LIN {X 0,Y 175.401,Z 600.795,A -85,B 0,C 180,E1 -24078.805,E2 -24078.805} C_VEL
LIN {X 0,Y 170.127,Z 592.607,A -85,B 0,C 180,E1 -24081.433,E2 -24081.433} C_VEL
LIN {X 0,Y 165.142,Z 585.432,A -85,B 0,C 180,E1 -24084.194,E2 -24084.194} C_VEL
LIN {X 0,Y 162.074,Z 581.252,A -85,B 0,C 180,E1 -24086.061,E2 -24086.061} C_VEL
LIN {X 0,Y 159.438,Z 578,A -85,B 0,C 180,E1 -24087.775,E2 -24087.775} C_VEL
LIN {X 0,Y 158.547,Z 576.618,A -85,B 0,C 180,E1 -24088.411,E2 -24088.411} C_VEL
LIN {X 0,Y 155.998,Z 573.951,A -85,B 0,C 180,E1 -24090.222,E2 -24090.222} C_VEL
LIN {X 0,Y 154.688,Z 571.494,A -85,B 0,C 180,E1 -24091.321,E2 -24091.321} C_VEL
LIN {X 0,Y 152.117,Z 569.719,A -85,B 0,C 180,E1 -24093.343,E2 -24093.343} C_VEL
LIN {X 0,Y 150.618,Z 567.322,A -85,B 0,C 180,E1 -24094.775,E2 -24094.775} C_VEL
LIN {X 0,Y 150.248,Z 565.769,A -85,B 0,C 180,E1 -24095.287,E2 -24095.287} C_VEL
LIN {X 0,Y 150.36,Z 565.755,A -85,B 0,C 180,E1 -24100.902,E2 -24100.902} C_VEL
LIN {X 0,Y 150.448,Z 565.742,A -85,B 0,C 180,E1 -24106.493,E2 -24106.493} C_VEL
LIN {X 0,Y 150.645,Z 565.698,A -85,B 0,C 180,E1 -24109.245,E2 -24109.245} C_VEL
LIN {X 0,Y 150.739,Z 565.693,A -85,B 0,C 180,E1 -24111.959,E2 -24111.959} C_VEL
LIN {X 0,Y 151.214,Z 565.649,A -85,B 0,C 180,E1 -24120,E2 -24120} C_VEL
LIN {X 0,Y 150.757,Z 565.696,A -85,B 0,C 180,E1 -24128.039,E2 -24128.039} C_VEL
LIN {X 0,Y 150.628,Z 565.705,A -85,B 0,C 180,E1 -24131.545,E2 -24131.545} C_VEL
LIN {X 0,Y 150.369,Z 565.735,A -85,B 0,C 180,E1 -24136.286,E2 -24136.286} C_VEL
LIN {X 0,Y 150.346,Z 565.743,A -85,B 0,C 180,E1 -24140.794,E2 -24140.794} C_VEL
LIN {X 0,Y 150.251,Z 565.771,A -85,B 0,C 180,E1 -24144.343,E2 -24144.343} C_VEL
LIN {X 0,Y 150.963,Z 568.144,A -85,B 0,C 180,E1 -24145.232,E2 -24145.232} C_VEL
LIN {X 0,Y 152.896,Z 570.41,A -85,B 0,C 180,E1 -24146.946,E2 -24146.946} C_VEL
LIN {X 0,Y 154.763,Z 571.667,A -85,B 0,C 180,E1 -24148.385,E2 -24148.385} C_VEL
LIN {X 0,Y 156.509,Z 574.692,A -85,B 0,C 180,E1 -24149.812,E2 -24149.812} C_VEL
LIN {X 0,Y 158.954,Z 577.113,A -85,B 0,C 180,E1 -24151.509,E2 -24151.509} C_VEL
LIN {X 0,Y 161.394,Z 580.608,A -85,B 0,C 180,E1 -24153.164,E2 -24153.164} C_VEL
LIN {X 0,Y 162.927,Z 582.356,A -85,B 0,C 180,E1 -24154.109,E2 -24154.109} C_VEL
LIN {X 0,Y 166.851,Z 588.676,A -85,B 0,C 180,E1 -24156.487,E2 -24156.487} C_VEL
LIN {X 0,Y 171.487,Z 596.616,A -85,B 0,C 180,E1 -24159.037,E2 -24159.037} C_VEL
LIN {X 0,Y 177.334,Z 608.087,A -85,B 0,C 180,E1 -24161.98,E2 -24161.98} C_VEL
LIN {X 0,Y 182.328,Z 619.835,A -85,B 0,C 180,E1 -24164.336,E2 -24164.336} C_VEL
LIN {X 0,Y 185.647,Z 628.738,A -85,B 0,C 180,E1 -24165.839,E2 -24165.839} C_VEL
LIN {X 0,Y 185.583,Z 633.595,A -85,B 0,C 180,E1 -24166.075,E2 -24166.075} C_VEL
LIN {X 0,Y 182.946,Z 673.813,A -85,B 0,C 180,E1 -24167.507,E2 -24167.507} C_VEL
LIN {X 0,Y 181.015,Z 687.597,A -85,B 0,C 180,E1 -24168.363,E2 -24168.363} C_VEL
LIN {X 0,Y 178.414,Z 699.716,A -85,B 0,C 180,E1 -24169.464,E2 -24169.464} C_VEL
LIN {X 0,Y 174.982,Z 712.384,A -85,B 0,C 180,E1 -24171.132,E2 -24171.132} C_VEL
LIN {X 0,Y 171.291,Z 723.647,A -85,B 0,C 180,E1 -24173.129,E2 -24173.129} C_VEL
LIN {X 0,Y 167.361,Z 733.791,A -85,B 0,C 180,E1 -24175.468,E2 -24175.468} C_VEL
LIN {X 0,Y 163.41,Z 742.938,A -85,B 0,C 180,E1 -24178.21,E2 -24178.21} C_VEL
LIN {X 0,Y 161.853,Z 746.354,A -85,B 0,C 180,E1 -24179.425,E2 -24179.425} C_VEL
LIN {X 0,Y 159.445,Z 750.159,A -85,B 0,C 180,E1 -24180.827,E2 -24180.827} C_VEL
LIN {X 0,Y 154.006,Z 755.881,A -85,B 0,C 180,E1 -24183.055,E2 -24183.055} C_VEL
LIN {X 0,Y 148.739,Z 760.905,A -85,B 0,C 180,E1 -24185.589,E2 -24185.589} C_VEL
LIN {X 0,Y 146.663,Z 763.652,A -85,B 0,C 180,E1 -24187.435,E2 -24187.435} C_VEL
LIN {X 0,Y 144.028,Z 768.399,A -85,B 0,C 180,E1 -24191.511,E2 -24191.511} C_VEL
LIN {X 0,Y 142.223,Z 772.01,A -85,B 0,C 180,E1 -24195.698,E2 -24195.698} C_VEL
LIN {X 0,Y 141.401,Z 773.873,A -85,B 0,C 180,E1 -24198.535,E2 -24198.535} C_VEL
LIN {X 0,Y 140.849,Z 775.27,A -85,B 0,C 180,E1 -24201.393,E2 -24201.393} C_VEL
LIN {X 0,Y 140.554,Z 776.27,A -85,B 0,C 180,E1 -24204.263,E2 -24204.263} C_VEL
LIN {X 0,Y 140.562,Z 777.087,A -85,B 0,C 180,E1 -24209.713,E2 -24209.713} C_VEL
LIN {X 0,Y 140.736,Z 776.871,A -85,B 0,C 180,E1 -24212.865,E2 -24212.865} C_VEL
LIN {X 0,Y 141.065,Z 776.256,A -85,B 0,C 180,E1 -24215.721,E2 -24215.721} C_VEL
LIN {X 0,Y 141.616,Z 775.252,A -85,B 0,C 180,E1 -24218.565,E2 -24218.565} C_VEL
LIN {X 0,Y 144.026,Z 772.019,A -85,B 0,C 180,E1 -24224.395,E2 -24224.395} C_VEL
LIN {X 0,Y 146.516,Z 776.665,A -85,B 0,C 180,E1 -24229.622,E2 -24229.622} C_VEL
LIN {X 0,Y 148.4,Z 778.596,A -85,B 0,C 180,E1 -24232.266,E2 -24232.266} C_VEL
LIN {X 0,Y 153.432,Z 781.157,A -85,B 0,C 180,E1 -24237.264,E2 -24237.264} C_VEL
LIN {X 0,Y 156.692,Z 781.963,A -85,B 0,C 180,E1 -24239.565,E2 -24239.565} C_VEL
LIN {X 0,Y 164.15,Z 782.273,A -85,B 0,C 180,E1 -24243.822,E2 -24243.822} C_VEL
LIN {X 0,Y 168.36,Z 781.919,A -85,B 0,C 180,E1 -24245.764,E2 -24245.764} C_VEL
LIN {X 0,Y 177.623,Z 779.864,A -85,B 0,C 180,E1 -24249.279,E2 -24249.279} C_VEL
LIN {X 0,Y 185.169,Z 777.289,A -85,B 0,C 180,E1 -24251.623,E2 -24251.623} C_VEL
LIN {X 0,Y 193.201,Z 773.68,A -85,B 0,C 180,E1 -24253.724,E2 -24253.724} C_VEL
LIN {X 0,Y 198.847,Z 770.696,A -85,B 0,C 180,E1 -24254.983,E2 -24254.983} C_VEL
LIN {X 0,Y 201.924,Z 768.865,A -85,B 0,C 180,E1 -24255.885,E2 -24255.885} C_VEL
LIN {X 0,Y 193.405,Z 773.579,A -85,B 0,C 180,E1 -24257.758,E2 -24257.758} C_VEL
LIN {X 0,Y 185.332,Z 777.13,A -85,B 0,C 180,E1 -24259.86,E2 -24259.86} C_VEL
LIN {X 0,Y 175.364,Z 780.219,A -85,B 0,C 180,E1 -24263.048,E2 -24263.048} C_VEL
LIN {X 0,Y 170.717,Z 781.07,A -85,B 0,C 180,E1 -24264.806,E2 -24264.806} C_VEL
LIN {X 0,Y 162.284,Z 781.531,A -85,B 0,C 180,E1 -24268.689,E2 -24268.689} C_VEL
LIN {X 0,Y 158.606,Z 781.187,A -85,B 0,C 180,E1 -24270.829,E2 -24270.829} C_VEL
LIN {X 0,Y 152.19,Z 779.18,A -85,B 0,C 180,E1 -24275.442,E2 -24275.442} C_VEL
LIN {X 0,Y 148.495,Z 776.67,A -85,B 0,C 180,E1 -24279.209,E2 -24279.209} C_VEL
LIN {X 0,Y 145.778,Z 773.203,A -85,B 0,C 180,E1 -24283.186,E2 -24283.186} C_VEL
LIN {X 0,Y 144.118,Z 768.862,A -85,B 0,C 180,E1 -24287.25,E2 -24287.25} C_VEL
LIN {X 0,Y 143.374,Z 764.179,A -85,B 0,C 180,E1 -24290.833,E2 -24290.833} C_VEL
LIN {X 0,Y 143.375,Z 757.493,A -85,B 0,C 180,E1 -24295.079,E2 -24295.079} C_VEL
LIN {X 0,Y 143.685,Z 750.494,A -85,B 0,C 180,E1 -24298.599,E2 -24298.599} C_VEL
LIN {X 0,Y 144.031,Z 742.449,A -85,B 0,C 180,E1 -24301.748,E2 -24301.748} C_VEL
LIN {X 0,Y 144.283,Z 733.555,A -85,B 0,C 180,E1 -24304.54,E2 -24304.54} C_VEL
LIN {X 0,Y 144.601,Z 723.972,A -85,B 0,C 180,E1 -24306.979,E2 -24306.979} C_VEL
LIN {X 0,Y 145.094,Z 712.443,A -85,B 0,C 180,E1 -24309.233,E2 -24309.233} C_VEL
LIN {X 0,Y 145.364,Z 701.518,A -85,B 0,C 180,E1 -24310.798,E2 -24310.798} C_VEL
LIN {X 0,Y 145.916,Z 666.157,A -85,B 0,C 180,E1 -24314.417,E2 -24314.417} C_VEL
LIN {X 0,Y 146.086,Z 645.484,A -85,B 0,C 180,E1 -24316.421,E2 -24316.421} C_VEL
LIN {X 0,Y 144.453,Z 621.674,A -85,B 0,C 180,E1 -24318.574,E2 -24318.574} C_VEL
LIN {X 0,Y 144.39,Z 617.741,A -85,B 0,C 180,E1 -24318.996,E2 -24318.996} C_VEL
LIN {X 0,Y 145.352,Z 604.834,A -85,B 0,C 180,E1 -24323.849,E2 -24323.849} C_VEL
LIN {X 0,Y 145.798,Z 602.705,A -85,B 0,C 180,E1 -24325.137,E2 -24325.137} C_VEL
LIN {X 0,Y 146.091,Z 602.477,A -85,B 0,C 180,E1 -24325.656,E2 -24325.656} C_VEL
LIN {X 0,Y 147.528,Z 602.404,A -85,B 0,C 180,E1 -24326.909,E2 -24326.909} C_VEL
LIN {X 0,Y 150.097,Z 600.201,A -85,B 0,C 180,E1 -24328.582,E2 -24328.582} C_VEL
LIN {X 0,Y 154.19,Z 595.325,A -85,B 0,C 180,E1 -24330.849,E2 -24330.849} C_VEL
LIN {X 0,Y 156.922,Z 595.505,A -85,B 0,C 180,E1 -24332.51,E2 -24332.51} C_VEL
LIN {X 0,Y 158.927,Z 594.524,A -85,B 0,C 180,E1 -24333.557,E2 -24333.557} C_VEL
LIN {X 0,Y 162.927,Z 594.201,A -85,B 0,C 180,E1 -24335.615,E2 -24335.615} C_VEL
LIN {X 0,Y 164.092,Z 594.078,A -85,B 0,C 180,E1 -24336.175,E2 -24336.175} C_VEL
LIN {X 0,Y 168.438,Z 600.642,A -85,B 0,C 180,E1 -24338.61,E2 -24338.61} C_VEL
LIN {X 0,Y 174.079,Z 610.004,A -85,B 0,C 180,E1 -24341.474,E2 -24341.474} C_VEL
LIN {X 0,Y 178.176,Z 617.897,A -85,B 0,C 180,E1 -24343.412,E2 -24343.412} C_VEL
LIN {X 0,Y 180.855,Z 624.585,A -85,B 0,C 180,E1 -24344.681,E2 -24344.681} C_VEL
LIN {X 0,Y 178.238,Z 663.283,A -85,B 0,C 180,E1 -24346.03,E2 -24346.03} C_VEL
LIN {X 0,Y 176.727,Z 676.165,A -85,B 0,C 180,E1 -24346.773,E2 -24346.773} C_VEL
LIN {X 0,Y 174.414,Z 688.968,A -85,B 0,C 180,E1 -24347.938,E2 -24347.938} C_VEL
LIN {X 0,Y 171.475,Z 700.769,A -85,B 0,C 180,E1 -24349.407,E2 -24349.407} C_VEL
LIN {X 0,Y 168.109,Z 711.495,A -85,B 0,C 180,E1 -24351.162,E2 -24351.162} C_VEL
LIN {X 0,Y 164.039,Z 722.429,A -85,B 0,C 180,E1 -24353.524,E2 -24353.524} C_VEL
LIN {X 0,Y 160.287,Z 731.314,A -85,B 0,C 180,E1 -24356.009,E2 -24356.009} C_VEL
LIN {X 0,Y 156.293,Z 739.948,A -85,B 0,C 180,E1 -24359.106,E2 -24359.106} C_VEL
LIN {X 0,Y 152.499,Z 747.445,A -85,B 0,C 180,E1 -24362.555,E2 -24362.555} C_VEL
LIN {X 0,Y 148.926,Z 753.853,A -85,B 0,C 180,E1 -24366.349,E2 -24366.349} C_VEL
LIN {X 0,Y 146.044,Z 758.933,A -85,B 0,C 180,E1 -24370.312,E2 -24370.312} C_VEL
LIN {X 0,Y 143.747,Z 762.872,A -85,B 0,C 180,E1 -24374.399,E2 -24374.399} C_VEL
LIN {X 0,Y 142.139,Z 765.777,A -85,B 0,C 180,E1 -24378.591,E2 -24378.591} C_VEL
LIN {X 0,Y 141.435,Z 767.165,A -85,B 0,C 180,E1 -24381.424,E2 -24381.424} C_VEL
LIN {X 0,Y 141.008,Z 768.151,A -85,B 0,C 180,E1 -24384.277,E2 -24384.277} C_VEL
LIN {X 0,Y 140.737,Z 768.758,A -85,B 0,C 180,E1 -24387.135,E2 -24387.135} C_VEL
LIN {X 0,Y 140.69,Z 768.984,A -85,B 0,C 180,E1 -24389.998,E2 -24389.998} C_VEL
LIN {X 0,Y 140.736,Z 768.789,A -85,B 0,C 180,E1 -24392.86,E2 -24392.86} C_VEL
LIN {X 0,Y 141.007,Z 768.204,A -85,B 0,C 180,E1 -24395.718,E2 -24395.718} C_VEL
LIN {X 0,Y 142.136,Z 765.884,A -85,B 0,C 180,E1 -24401.405,E2 -24401.405} C_VEL
LIN {X 0,Y 143.73,Z 763.013,A -85,B 0,C 180,E1 -24405.598,E2 -24405.598} C_VEL
LIN {X 0,Y 145.977,Z 759.117,A -85,B 0,C 180,E1 -24409.692,E2 -24409.692} C_VEL
LIN {X 0,Y 148.832,Z 754.096,A -85,B 0,C 180,E1 -24413.662,E2 -24413.662} C_VEL
LIN {X 0,Y 152.426,Z 747.763,A -85,B 0,C 180,E1 -24417.454,E2 -24417.454} C_VEL
LIN {X 0,Y 156.142,Z 740.567,A -85,B 0,C 180,E1 -24420.801,E2 -24420.801} C_VEL
LIN {X 0,Y 160.206,Z 731.769,A -85,B 0,C 180,E1 -24424.006,E2 -24424.006} C_VEL
LIN {X 0,Y 164.362,Z 721.91,A -85,B 0,C 180,E1 -24426.769,E2 -24426.769} C_VEL
LIN {X 0,Y 168.516,Z 710.802,A -85,B 0,C 180,E1 -24429.105,E2 -24429.105} C_VEL
LIN {X 0,Y 171.87,Z 699.908,A -85,B 0,C 180,E1 -24430.861,E2 -24430.861} C_VEL
LIN {X 0,Y 174.791,Z 687.856,A -85,B 0,C 180,E1 -24432.334,E2 -24432.334} C_VEL
LIN {X 0,Y 177.054,Z 675.297,A -85,B 0,C 180,E1 -24433.42,E2 -24433.42} C_VEL
LIN {X 0,Y 178.514,Z 662.659,A -85,B 0,C 180,E1 -24434.119,E2 -24434.119} C_VEL
LIN {X 0,Y 181.017,Z 624.787,A -85,B 0,C 180,E1 -24435.451,E2 -24435.451} C_VEL
LIN {X 0,Y 177.262,Z 615.769,A -85,B 0,C 180,E1 -24437.232,E2 -24437.232} C_VEL
LIN {X 0,Y 171.522,Z 605.541,A -85,B 0,C 180,E1 -24440.013,E2 -24440.013} C_VEL
LIN {X 0,Y 166.095,Z 596.948,A -85,B 0,C 180,E1 -24442.917,E2 -24442.917} C_VEL
LIN {X 0,Y 161.753,Z 590.618,A -85,B 0,C 180,E1 -24445.502,E2 -24445.502} C_VEL
LIN {X 0,Y 159.087,Z 586.942,A -85,B 0,C 180,E1 -24447.236,E2 -24447.236} C_VEL
LIN {X 0,Y 156.431,Z 583.249,A -85,B 0,C 180,E1 -24449.115,E2 -24449.115} C_VEL
LIN {X 0,Y 153.386,Z 579.692,A -85,B 0,C 180,E1 -24451.429,E2 -24451.429} C_VEL
LIN {X 0,Y 152.306,Z 577.95,A -85,B 0,C 180,E1 -24452.364,E2 -24452.364} C_VEL
LIN {X 0,Y 149.696,Z 575.629,A -85,B 0,C 180,E1 -24454.609,E2 -24454.609} C_VEL
LIN {X 0,Y 148.169,Z 572.834,A -85,B 0,C 180,E1 -24456.223,E2 -24456.223} C_VEL
LIN {X 0,Y 147.867,Z 572.411,A -85,B 0,C 180,E1 -24456.543,E2 -24456.543} C_VEL
LIN {X 0,Y 145.469,Z 570.902,A -85,B 0,C 180,E1 -24459.052,E2 -24459.052} C_VEL
LIN {X 0,Y 143.833,Z 568.534,A -85,B 0,C 180,E1 -24461.205,E2 -24461.205} C_VEL
LIN {X 0,Y 143.277,Z 566.62,A -85,B 0,C 180,E1 -24462.331,E2 -24462.331} C_VEL
LIN {X 0,Y 143.588,Z 566.58,A -85,B 0,C 180,E1 -24468.709,E2 -24468.709} C_VEL
LIN {X 0,Y 143.659,Z 566.571,A -85,B 0,C 180,E1 -24471.56,E2 -24471.56} C_VEL
LIN {X 0,Y 144.172,Z 566.526,A -85,B 0,C 180,E1 -24480,E2 -24480} C_VEL
LIN {X 0,Y 143.679,Z 566.573,A -85,B 0,C 180,E1 -24488.438,E2 -24488.438} C_VEL
LIN {X 0,Y 143.565,Z 566.586,A -85,B 0,C 180,E1 -24491.758,E2 -24491.758} C_VEL
LIN {X 0,Y 143.287,Z 566.71,A -85,B 0,C 180,E1 -24497.483,E2 -24497.483} C_VEL
LIN {X 0,Y 143.994,Z 568.91,A -85,B 0,C 180,E1 -24498.681,E2 -24498.681} C_VEL
LIN {X 0,Y 145.834,Z 571.244,A -85,B 0,C 180,E1 -24501.008,E2 -24501.008} C_VEL
LIN {X 0,Y 148.092,Z 572.649,A -85,B 0,C 180,E1 -24503.326,E2 -24503.326} C_VEL
LIN {X 0,Y 149.662,Z 575.608,A -85,B 0,C 180,E1 -24505.001,E2 -24505.001} C_VEL
LIN {X 0,Y 152.592,Z 578.316,A -85,B 0,C 180,E1 -24507.517,E2 -24507.517} C_VEL
LIN {X 0,Y 154.86,Z 581.681,A -85,B 0,C 180,E1 -24509.387,E2 -24509.387} C_VEL
LIN {X 0,Y 156.547,Z 583.501,A -85,B 0,C 180,E1 -24510.618,E2 -24510.618} C_VEL
LIN {X 0,Y 159.281,Z 587.171,A -85,B 0,C 180,E1 -24512.531,E2 -24512.531} C_VEL
LIN {X 0,Y 161.27,Z 590.153,A -85,B 0,C 180,E1 -24513.848,E2 -24513.848} C_VEL
LIN {X 0,Y 165.359,Z 596.983,A -85,B 0,C 180,E1 -24516.384,E2 -24516.384} C_VEL
LIN {X 0,Y 170.544,Z 606.852,A -85,B 0,C 180,E1 -24519.316,E2 -24519.316} C_VEL
LIN {X 0,Y 175.099,Z 616.732,A -85,B 0,C 180,E1 -24521.689,E2 -24521.689} C_VEL
LIN {X 0,Y 179.891,Z 629.091,A -85,B 0,C 180,E1 -24524.062,E2 -24524.062} C_VEL
LIN {X 0,Y 180.657,Z 631.538,A -85,B 0,C 180,E1 -24524.447,E2 -24524.447} C_VEL
LIN {X 0,Y 177.817,Z 673.249,A -85,B 0,C 180,E1 -24525.942,E2 -24525.942} C_VEL
LIN {X 0,Y 175.897,Z 686.736,A -85,B 0,C 180,E1 -24526.778,E2 -24526.778} C_VEL
LIN {X 0,Y 173.072,Z 699.517,A -85,B 0,C 180,E1 -24527.934,E2 -24527.934} C_VEL
LIN {X 0,Y 169.524,Z 712.185,A -85,B 0,C 180,E1 -24529.629,E2 -24529.629} C_VEL
LIN {X 0,Y 165.651,Z 723.445,A -85,B 0,C 180,E1 -24531.651,E2 -24531.651} C_VEL
LIN {X 0,Y 161.561,Z 733.589,A -85,B 0,C 180,E1 -24534.04,E2 -24534.04} C_VEL
LIN {X 0,Y 157.396,Z 742.735,A -85,B 0,C 180,E1 -24536.843,E2 -24536.843} C_VEL
LIN {X 0,Y 153.054,Z 751.658,A -85,B 0,C 180,E1 -24540.425,E2 -24540.425} C_VEL
LIN {X 0,Y 149.376,Z 758.839,A -85,B 0,C 180,E1 -24544.205,E2 -24544.205} C_VEL
LIN {X 0,Y 146.663,Z 763.652,A -85,B 0,C 180,E1 -24547.435,E2 -24547.435} C_VEL
LIN {X 0,Y 144.699,Z 766.223,A -85,B 0,C 180,E1 -24549.379,E2 -24549.379} C_VEL
LIN {X 0,Y 140.003,Z 769.828,A -85,B 0,C 180,E1 -24552.585,E2 -24552.585} C_VEL
LIN {X 0,Y 135.651,Z 772.625,A -85,B 0,C 180,E1 -24556.113,E2 -24556.113} C_VEL
LIN {X 0,Y 134.292,Z 773.932,A -85,B 0,C 180,E1 -24558.496,E2 -24558.496} C_VEL
LIN {X 0,Y 133.47,Z 776.065,A -85,B 0,C 180,E1 -24563.957,E2 -24563.957} C_VEL
LIN {X 0,Y 133.397,Z 776.676,A -85,B 0,C 180,E1 -24566.983,E2 -24566.983} C_VEL
LIN {X 0,Y 133.495,Z 776.89,A -85,B 0,C 180,E1 -24570.003,E2 -24570.003} C_VEL
LIN {X 0,Y 133.659,Z 776.666,A -85,B 0,C 180,E1 -24573.017,E2 -24573.017} C_VEL
LIN {X 0,Y 134.02,Z 776.052,A -85,B 0,C 180,E1 -24576.023,E2 -24576.023} C_VEL
LIN {X 0,Y 135.611,Z 773.645,A -85,B 0,C 180,E1 -24581.967,E2 -24581.967} C_VEL
LIN {X 0,Y 137.874,Z 771.009,A -85,B 0,C 180,E1 -24586.189,E2 -24586.189} C_VEL
LIN {X 0,Y 140.986,Z 776.112,A -85,B 0,C 180,E1 -24591.957,E2 -24591.957} C_VEL
LIN {X 0,Y 144.36,Z 778.88,A -85,B 0,C 180,E1 -24595.989,E2 -24595.989} C_VEL
LIN {X 0,Y 147.212,Z 780.224,A -85,B 0,C 180,E1 -24598.519,E2 -24598.519} C_VEL
LIN {X 0,Y 154.296,Z 781.974,A -85,B 0,C 180,E1 -24603.135,E2 -24603.135} C_VEL
LIN {X 0,Y 162.659,Z 782.115,A -85,B 0,C 180,E1 -24607.224,E2 -24607.224} C_VEL
LIN {X 0,Y 167.305,Z 781.708,A -85,B 0,C 180,E1 -24609.06,E2 -24609.06} C_VEL
LIN {X 0,Y 177.326,Z 779.544,A -85,B 0,C 180,E1 -24612.36,E2 -24612.36} C_VEL
LIN {X 0,Y 185.417,Z 776.888,A -85,B 0,C 180,E1 -24614.527,E2 -24614.527} C_VEL
LIN {X 0,Y 189.41,Z 775.374,A -85,B 0,C 180,E1 -24615.448,E2 -24615.448} C_VEL
LIN {X 0,Y 190.285,Z 774.982,A -85,B 0,C 180,E1 -24615.896,E2 -24615.896} C_VEL
LIN {X 0,Y 180.019,Z 778.686,A -85,B 0,C 180,E1 -24618.418,E2 -24618.418} C_VEL
LIN {X 0,Y 173.107,Z 780.424,A -85,B 0,C 180,E1 -24620.481,E2 -24620.481} C_VEL
LIN {X 0,Y 164.969,Z 781.51,A -85,B 0,C 180,E1 -24623.386,E2 -24623.386} C_VEL
LIN {X 0,Y 160.459,Z 781.691,A -85,B 0,C 180,E1 -24625.292,E2 -24625.292} C_VEL
LIN {X 0,Y 156.274,Z 781.365,A -85,B 0,C 180,E1 -24627.339,E2 -24627.339} C_VEL
LIN {X 0,Y 149.005,Z 779.659,A -85,B 0,C 180,E1 -24631.858,E2 -24631.858} C_VEL
LIN {X 0,Y 145.834,Z 778.186,A -85,B 0,C 180,E1 -24634.296,E2 -24634.296} C_VEL
LIN {X 0,Y 140.947,Z 774.058,A -85,B 0,C 180,E1 -24639.572,E2 -24639.572} C_VEL
LIN {X 0,Y 138.554,Z 769.895,A -85,B 0,C 180,E1 -24643.801,E2 -24643.801} C_VEL
LIN {X 0,Y 137.248,Z 764.668,A -85,B 0,C 180,E1 -24648.181,E2 -24648.181} C_VEL
LIN {X 0,Y 136.795,Z 759.388,A -85,B 0,C 180,E1 -24651.878,E2 -24651.878} C_VEL
LIN {X 0,Y 136.987,Z 752.975,A -85,B 0,C 180,E1 -24655.587,E2 -24655.587} C_VEL
LIN {X 0,Y 137.336,Z 745.098,A -85,B 0,C 180,E1 -24659.267,E2 -24659.267} C_VEL
LIN {X 0,Y 137.55,Z 735.876,A -85,B 0,C 180,E1 -24662.563,E2 -24662.563} C_VEL
LIN {X 0,Y 137.824,Z 726.826,A -85,B 0,C 180,E1 -24665.12,E2 -24665.12} C_VEL
LIN {X 0,Y 138.21,Z 715.513,A -85,B 0,C 180,E1 -24667.671,E2 -24667.671} C_VEL
LIN {X 0,Y 138.601,Z 703.296,A -85,B 0,C 180,E1 -24669.67,E2 -24669.67} C_VEL
LIN {X 0,Y 138.892,Z 674.77,A -85,B 0,C 180,E1 -24672.883,E2 -24672.883} C_VEL
LIN {X 0,Y 139.087,Z 645.414,A -85,B 0,C 180,E1 -24675.911,E2 -24675.911} C_VEL
LIN {X 0,Y 137.588,Z 625.741,A -85,B 0,C 180,E1 -24677.847,E2 -24677.847} C_VEL
LIN {X 0,Y 137.357,Z 621.52,A -85,B 0,C 180,E1 -24678.65,E2 -24678.65} C_VEL
LIN {X 0,Y 137.478,Z 619.579,A -85,B 0,C 180,E1 -24679.408,E2 -24679.408} C_VEL
LIN {X 0,Y 139.105,Z 618.541,A -85,B 0,C 180,E1 -24681.26,E2 -24681.26} C_VEL
LIN {X 0,Y 141.733,Z 615.09,A -85,B 0,C 180,E1 -24683.439,E2 -24683.439} C_VEL
LIN {X 0,Y 145.381,Z 609.569,A -85,B 0,C 180,E1 -24685.983,E2 -24685.983} C_VEL
LIN {X 0,Y 147.798,Z 609.114,A -85,B 0,C 180,E1 -24687.814,E2 -24687.814} C_VEL
LIN {X 0,Y 150.901,Z 606.575,A -85,B 0,C 180,E1 -24689.751,E2 -24689.751} C_VEL
LIN {X 0,Y 154.328,Z 602.625,A -85,B 0,C 180,E1 -24691.581,E2 -24691.581} C_VEL
LIN {X 0,Y 157.165,Z 602.339,A -85,B 0,C 180,E1 -24693.216,E2 -24693.216} C_VEL
LIN {X 0,Y 159.182,Z 601.585,A -85,B 0,C 180,E1 -24694.258,E2 -24694.258} C_VEL
LIN {X 0,Y 162.326,Z 601.517,A -85,B 0,C 180,E1 -24695.863,E2 -24695.863} C_VEL
LIN {X 0,Y 168.534,Z 611.78,A -85,B 0,C 180,E1 -24699.393,E2 -24699.393} C_VEL
LIN {X 0,Y 173.632,Z 621.335,A -85,B 0,C 180,E1 -24701.999,E2 -24701.999} C_VEL
LIN {X 0,Y 175.806,Z 626.839,A -85,B 0,C 180,E1 -24703.111,E2 -24703.111} C_VEL
LIN {X 0,Y 173.101,Z 664.64,A -85,B 0,C 180,E1 -24704.445,E2 -24704.445} C_VEL
LIN {X 0,Y 171.437,Z 677.509,A -85,B 0,C 180,E1 -24705.241,E2 -24705.241} C_VEL
LIN {X 0,Y 168.973,Z 690.307,A -85,B 0,C 180,E1 -24706.456,E2 -24706.456} C_VEL
LIN {X 0,Y 166.154,Z 700.979,A -85,B 0,C 180,E1 -24707.816,E2 -24707.816} C_VEL
LIN {X 0,Y 162.651,Z 711.704,A -85,B 0,C 180,E1 -24709.596,E2 -24709.596} C_VEL
LIN {X 0,Y 158.393,Z 722.637,A -85,B 0,C 180,E1 -24711.999,E2 -24711.999} C_VEL
LIN {X 0,Y 154.442,Z 731.52,A -85,B 0,C 180,E1 -24714.533,E2 -24714.533} C_VEL
LIN {X 0,Y 150.112,Z 740.401,A -85,B 0,C 180,E1 -24717.815,E2 -24717.815} C_VEL
LIN {X 0,Y 146.245,Z 747.651,A -85,B 0,C 180,E1 -24721.275,E2 -24721.275} C_VEL
LIN {X 0,Y 142.435,Z 754.06,A -85,B 0,C 180,E1 -24725.201,E2 -24725.201} C_VEL
LIN {X 0,Y 139.367,Z 759.139,A -85,B 0,C 180,E1 -24729.327,E2 -24729.327} C_VEL
LIN {X 0,Y 136.918,Z 763.078,A -85,B 0,C 180,E1 -24733.599,E2 -24733.599} C_VEL
LIN {X 0,Y 135.175,Z 765.983,A -85,B 0,C 180,E1 -24737.994,E2 -24737.994} C_VEL
LIN {X 0,Y 134.429,Z 767.37,A -85,B 0,C 180,E1 -24740.974,E2 -24740.974} C_VEL
LIN {X 0,Y 133.95,Z 768.356,A -85,B 0,C 180,E1 -24743.974,E2 -24743.974} C_VEL
LIN {X 0,Y 133.596,Z 769.099,A -85,B 0,C 180,E1 -24748.24,E2 -24748.24} C_VEL
LIN {X 0,Y 133.659,Z 768.993,A -85,B 0,C 180,E1 -24753.011,E2 -24753.011} C_VEL
LIN {X 0,Y 133.948,Z 768.409,A -85,B 0,C 180,E1 -24756.021,E2 -24756.021} C_VEL
LIN {X 0,Y 135.171,Z 766.089,A -85,B 0,C 180,E1 -24762.001,E2 -24762.001} C_VEL
LIN {X 0,Y 136.901,Z 763.217,A -85,B 0,C 180,E1 -24766.398,E2 -24766.398} C_VEL
LIN {X 0,Y 139.306,Z 759.321,A -85,B 0,C 180,E1 -24770.677,E2 -24770.677} C_VEL
LIN {X 0,Y 142.347,Z 754.299,A -85,B 0,C 180,E1 -24774.81,E2 -24774.81} C_VEL
LIN {X 0,Y 146.163,Z 747.966,A -85,B 0,C 180,E1 -24778.737,E2 -24778.737} C_VEL
LIN {X 0,Y 150.678,Z 739.542,A -85,B 0,C 180,E1 -24782.705,E2 -24782.705} C_VEL
LIN {X 0,Y 155.212,Z 730.193,A -85,B 0,C 180,E1 -24786.058,E2 -24786.058} C_VEL
LIN {X 0,Y 159.213,Z 721.007,A -85,B 0,C 180,E1 -24788.57,E2 -24788.57} C_VEL
LIN {X 0,Y 163.58,Z 709.58,A -85,B 0,C 180,E1 -24790.931,E2 -24790.931} C_VEL
LIN {X 0,Y 167.077,Z 698.344,A -85,B 0,C 180,E1 -24792.707,E2 -24792.707} C_VEL
LIN {X 0,Y 169.9,Z 686.909,A -85,B 0,C 180,E1 -24794.06,E2 -24794.06} C_VEL
LIN {X 0,Y 172.153,Z 674.217,A -85,B 0,C 180,E1 -24795.128,E2 -24795.128} C_VEL
LIN {X 0,Y 173.683,Z 660.772,A -85,B 0,C 180,E1 -24795.829,E2 -24795.829} C_VEL
LIN {X 0,Y 175.972,Z 627.04,A -85,B 0,C 180,E1 -24797.024,E2 -24797.024} C_VEL
LIN {X 0,Y 172.933,Z 619.726,A -85,B 0,C 180,E1 -24798.572,E2 -24798.572} C_VEL
LIN {X 0,Y 167.752,Z 610.369,A -85,B 0,C 180,E1 -24801.258,E2 -24801.258} C_VEL
LIN {X 0,Y 162.205,Z 601.206,A -85,B 0,C 180,E1 -24804.467,E2 -24804.467} C_VEL
LIN {X 0,Y 156.679,Z 593.188,A -85,B 0,C 180,E1 -24808.103,E2 -24808.103} C_VEL
LIN {X 0,Y 153.194,Z 588.558,A -85,B 0,C 180,E1 -24810.714,E2 -24810.714} C_VEL
LIN {X 0,Y 150.501,Z 584.837,A -85,B 0,C 180,E1 -24812.995,E2 -24812.995} C_VEL
LIN {X 0,Y 147.145,Z 581.165,A -85,B 0,C 180,E1 -24816.141,E2 -24816.141} C_VEL
LIN {X 0,Y 146.081,Z 579.154,A -85,B 0,C 180,E1 -24817.363,E2 -24817.363} C_VEL
LIN {X 0,Y 143.353,Z 576.977,A -85,B 0,C 180,E1 -24820.489,E2 -24820.489} C_VEL
LIN {X 0,Y 141.734,Z 573.898,A -85,B 0,C 180,E1 -24822.97,E2 -24822.97} C_VEL
LIN {X 0,Y 141.469,Z 573.476,A -85,B 0,C 180,E1 -24823.402,E2 -24823.402} C_VEL
LIN {X 0,Y 138.7,Z 571.786,A -85,B 0,C 180,E1 -24828.306,E2 -24828.306} C_VEL
LIN {X 0,Y 136.716,Z 568.001,A -85,B 0,C 180,E1 -24835.762,E2 -24835.762} C_VEL
LIN {X 0,Y 136.723,Z 567.429,A -85,B 0,C 180,E1 -24836.685,E2 -24836.685} C_VEL
LIN {X 0,Y 137.129,Z 567.403,A -85,B 0,C 180,E1 -24840,E2 -24840} C_VEL
LIN {X 0,Y 136.712,Z 567.538,A -85,B 0,C 180,E1 -24843.5,E2 -24843.5} C_VEL
LIN {X 0,Y 137.235,Z 569.712,A -85,B 0,C 180,E1 -24846.986,E2 -24846.986} C_VEL
LIN {X 0,Y 140.336,Z 573.047,A -85,B 0,C 180,E1 -24854.501,E2 -24854.501} C_VEL
LIN {X 0,Y 141.681,Z 573.747,A -85,B 0,C 180,E1 -24856.572,E2 -24856.572} C_VEL
LIN {X 0,Y 143.097,Z 576.623,A -85,B 0,C 180,E1 -24858.802,E2 -24858.802} C_VEL
LIN {X 0,Y 145.487,Z 578.849,A -85,B 0,C 180,E1 -24861.663,E2 -24861.663} C_VEL
LIN {X 0,Y 146.238,Z 579.435,A -85,B 0,C 180,E1 -24862.46,E2 -24862.46} C_VEL
LIN {X 0,Y 148.311,Z 582.736,A -85,B 0,C 180,E1 -24864.683,E2 -24864.683} C_VEL
LIN {X 0,Y 150.439,Z 584.806,A -85,B 0,C 180,E1 -24866.594,E2 -24866.594} C_VEL
LIN {X 0,Y 153.062,Z 588.426,A -85,B 0,C 180,E1 -24868.824,E2 -24868.824} C_VEL
LIN {X 0,Y 154.299,Z 589.992,A -85,B 0,C 180,E1 -24869.786,E2 -24869.786} C_VEL
LIN {X 0,Y 157.717,Z 594.695,A -85,B 0,C 180,E1 -24872.267,E2 -24872.267} C_VEL
LIN {X 0,Y 162.367,Z 602.857,A -85,B 0,C 180,E1 -24875.376,E2 -24875.376} C_VEL
LIN {X 0,Y 167.286,Z 612.629,A -85,B 0,C 180,E1 -24878.334,E2 -24878.334} C_VEL
LIN {X 0,Y 171.497,Z 622.324,A -85,B 0,C 180,E1 -24880.681,E2 -24880.681} C_VEL
LIN {X 0,Y 175.614,Z 633.497,A -85,B 0,C 180,E1 -24882.87,E2 -24882.87} C_VEL
LIN {X 0,Y 172.728,Z 673.511,A -85,B 0,C 180,E1 -24884.326,E2 -24884.326} C_VEL
LIN {X 0,Y 170.747,Z 686.804,A -85,B 0,C 180,E1 -24885.167,E2 -24885.167} C_VEL
LIN {X 0,Y 167.876,Z 699.319,A -85,B 0,C 180,E1 -24886.313,E2 -24886.313} C_VEL
LIN {X 0,Y 164.191,Z 711.985,A -85,B 0,C 180,E1 -24888.028,E2 -24888.028} C_VEL
LIN {X 0,Y 160.131,Z 723.244,A -85,B 0,C 180,E1 -24890.071,E2 -24890.071} C_VEL
LIN {X 0,Y 155.856,Z 733.387,A -85,B 0,C 180,E1 -24892.504,E2 -24892.504} C_VEL
LIN {X 0,Y 151.491,Z 742.533,A -85,B 0,C 180,E1 -24895.371,E2 -24895.371} C_VEL
LIN {X 0,Y 146.823,Z 751.589,A -85,B 0,C 180,E1 -24899.114,E2 -24899.114} C_VEL
LIN {X 0,Y 142.999,Z 758.637,A -85,B 0,C 180,E1 -24902.964,E2 -24902.964} C_VEL
LIN {X 0,Y 139.863,Z 763.819,A -85,B 0,C 180,E1 -24906.614,E2 -24906.614} C_VEL
LIN {X 0,Y 137.28,Z 768.194,A -85,B 0,C 180,E1 -24910.566,E2 -24910.566} C_VEL
LIN {X 0,Y 135.33,Z 771.806,A -85,B 0,C 180,E1 -24914.953,E2 -24914.953} C_VEL
LIN {X 0,Y 134.292,Z 773.932,A -85,B 0,C 180,E1 -24918.496,E2 -24918.496} C_VEL
LIN {X 0,Y 133.144,Z 775.073,A -85,B 0,C 180,E1 -24920.94,E2 -24920.94} C_VEL
LIN {X 0,Y 129.888,Z 776.267,A -85,B 0,C 180,E1 -24924.99,E2 -24924.99} C_VEL
LIN {X 0,Y 127.431,Z 776.641,A -85,B 0,C 180,E1 -24928.377,E2 -24928.377} C_VEL
LIN {X 0,Y 126.5,Z 776.64,A -85,B 0,C 180,E1 -24931.038,E2 -24931.038} C_VEL
LIN {X 0,Y 126.474,Z 776.55,A -85,B 0,C 180,E1 -24931.938,E2 -24931.938} C_VEL
LIN {X 0,Y 126.969,Z 775.847,A -85,B 0,C 180,E1 -24936.359,E2 -24936.359} C_VEL
LIN {X 0,Y 128.685,Z 773.44,A -85,B 0,C 180,E1 -24942.621,E2 -24942.621} C_VEL
LIN {X 0,Y 131.871,Z 769.901,A -85,B 0,C 180,E1 -24948.149,E2 -24948.149} C_VEL
LIN {X 0,Y 135.72,Z 775.414,A -85,B 0,C 180,E1 -24954.476,E2 -24954.476} C_VEL
LIN {X 0,Y 141.109,Z 779.05,A -85,B 0,C 180,E1 -24959.874,E2 -24959.874} C_VEL
LIN {X 0,Y 144.586,Z 780.397,A -85,B 0,C 180,E1 -24962.325,E2 -24962.325} C_VEL
LIN {X 0,Y 152.601,Z 781.923,A -85,B 0,C 180,E1 -24966.78,E2 -24966.78} C_VEL
LIN {X 0,Y 157.074,Z 782.157,A -85,B 0,C 180,E1 -24968.788,E2 -24968.788} C_VEL
LIN {X 0,Y 166.923,Z 781.5,A -85,B 0,C 180,E1 -24972.352,E2 -24972.352} C_VEL
LIN {X 0,Y 172.187,Z 780.594,A -85,B 0,C 180,E1 -24973.94,E2 -24973.94} C_VEL
LIN {X 0,Y 177.681,Z 779.268,A -85,B 0,C 180,E1 -24975.398,E2 -24975.398} C_VEL
LIN {X 0,Y 177.957,Z 779.184,A -85,B 0,C 180,E1 -24976.079,E2 -24976.079} C_VEL
LIN {X 0,Y 168.213,Z 781.135,A -85,B 0,C 180,E1 -24978.77,E2 -24978.77} C_VEL
LIN {X 0,Y 159.322,Z 781.796,A -85,B 0,C 180,E1 -24981.861,E2 -24981.861} C_VEL
LIN {X 0,Y 150.364,Z 780.939,A -85,B 0,C 180,E1 -24985.883,E2 -24985.883} C_VEL
LIN {X 0,Y 146.432,Z 780.03,A -85,B 0,C 180,E1 -24988.133,E2 -24988.133} C_VEL
LIN {X 0,Y 139.601,Z 776.859,A -85,B 0,C 180,E1 -24993.058,E2 -24993.058} C_VEL
LIN {X 0,Y 135.662,Z 773.544,A -85,B 0,C 180,E1 -24997.136,E2 -24997.136} C_VEL
LIN {X 0,Y 132.807,Z 769.267,A -85,B 0,C 180,E1 -25001.488,E2 -25001.488} C_VEL
LIN {X 0,Y 131.044,Z 763.829,A -85,B 0,C 180,E1 -25006.206,E2 -25006.206} C_VEL
LIN {X 0,Y 130.363,Z 756.382,A -85,B 0,C 180,E1 -25011.474,E2 -25011.474} C_VEL
LIN {X 0,Y 130.569,Z 749.516,A -85,B 0,C 180,E1 -25015.369,E2 -25015.369} C_VEL
LIN {X 0,Y 130.909,Z 742.762,A -85,B 0,C 180,E1 -25018.462,E2 -25018.462} C_VEL
LIN {X 0,Y 131.042,Z 735.507,A -85,B 0,C 180,E1 -25021.153,E2 -25021.153} C_VEL
LIN {X 0,Y 131.23,Z 726.66,A -85,B 0,C 180,E1 -25023.839,E2 -25023.839} C_VEL
LIN {X 0,Y 131.51,Z 715.476,A -85,B 0,C 180,E1 -25026.521,E2 -25026.521} C_VEL
LIN {X 0,Y 131.866,Z 703.333,A -85,B 0,C 180,E1 -25028.621,E2 -25028.621} C_VEL
LIN {X 0,Y 132.054,Z 674.348,A -85,B 0,C 180,E1 -25032.097,E2 -25032.097} C_VEL
LIN {X 0,Y 132.159,Z 649.998,A -85,B 0,C 180,E1 -25034.927,E2 -25034.927} C_VEL
LIN {X 0,Y 132.119,Z 646.574,A -85,B 0,C 180,E1 -25035.58,E2 -25035.58} C_VEL
LIN {X 0,Y 131.948,Z 644.924,A -85,B 0,C 180,E1 -25036.265,E2 -25036.265} C_VEL
LIN {X 0,Y 132.008,Z 644.66,A -85,B 0,C 180,E1 -25036.595,E2 -25036.595} C_VEL
LIN {X 0,Y 132.598,Z 644.365,A -85,B 0,C 180,E1 -25037.431,E2 -25037.431} C_VEL
LIN {X 0,Y 133.522,Z 642.268,A -85,B 0,C 180,E1 -25038.316,E2 -25038.316} C_VEL
LIN {X 0,Y 135.014,Z 637.25,A -85,B 0,C 180,E1 -25039.381,E2 -25039.381} C_VEL
LIN {X 0,Y 137.852,Z 626.151,A -85,B 0,C 180,E1 -25040.986,E2 -25040.986} C_VEL
LIN {X 0,Y 139.757,Z 624.654,A -85,B 0,C 180,E1 -25042.762,E2 -25042.762} C_VEL
LIN {X 0,Y 143.021,Z 620.467,A -85,B 0,C 180,E1 -25045.247,E2 -25045.247} C_VEL
LIN {X 0,Y 145.566,Z 616.713,A -85,B 0,C 180,E1 -25046.913,E2 -25046.913} C_VEL
LIN {X 0,Y 148.462,Z 615.591,A -85,B 0,C 180,E1 -25048.946,E2 -25048.946} C_VEL
LIN {X 0,Y 152.03,Z 612.684,A -85,B 0,C 180,E1 -25051.05,E2 -25051.05} C_VEL
LIN {X 0,Y 154.992,Z 609.618,A -85,B 0,C 180,E1 -25052.579,E2 -25052.579} C_VEL
LIN {X 0,Y 157.941,Z 608.975,A -85,B 0,C 180,E1 -25054.18,E2 -25054.18} C_VEL
LIN {X 0,Y 160.209,Z 608.712,A -85,B 0,C 180,E1 -25055.346,E2 -25055.346} C_VEL
LIN {X 0,Y 166.088,Z 618.853,A -85,B 0,C 180,E1 -25058.828,E2 -25058.828} C_VEL
LIN {X 0,Y 169.957,Z 626.668,A -85,B 0,C 180,E1 -25060.932,E2 -25060.932} C_VEL
LIN {X 0,Y 170.888,Z 629.161,A -85,B 0,C 180,E1 -25061.45,E2 -25061.45} C_VEL
LIN {X 0,Y 168.182,Z 665.178,A -85,B 0,C 180,E1 -25062.735,E2 -25062.735} C_VEL
LIN {X 0,Y 166.422,Z 678.102,A -85,B 0,C 180,E1 -25063.557,E2 -25063.557} C_VEL
LIN {X 0,Y 163.638,Z 691.646,A -85,B 0,C 180,E1 -25064.872,E2 -25064.872} C_VEL
LIN {X 0,Y 160.464,Z 702.914,A -85,B 0,C 180,E1 -25066.382,E2 -25066.382} C_VEL
LIN {X 0,Y 156.3,Z 714.537,A -85,B 0,C 180,E1 -25068.451,E2 -25068.451} C_VEL
LIN {X 0,Y 151.899,Z 724.977,A -85,B 0,C 180,E1 -25070.918,E2 -25070.918} C_VEL
LIN {X 0,Y 147.855,Z 733.501,A -85,B 0,C 180,E1 -25073.544,E2 -25073.544} C_VEL
LIN {X 0,Y 143.879,Z 741.109,A -85,B 0,C 180,E1 -25076.523,E2 -25076.523} C_VEL
LIN {X 0,Y 140.074,Z 747.858,A -85,B 0,C 180,E1 -25079.882,E2 -25079.882} C_VEL
LIN {X 0,Y 136.011,Z 754.267,A -85,B 0,C 180,E1 -25083.944,E2 -25083.944} C_VEL
LIN {X 0,Y 132.742,Z 759.345,A -85,B 0,C 180,E1 -25088.244,E2 -25088.244} C_VEL
LIN {X 0,Y 130.108,Z 763.284,A -85,B 0,C 180,E1 -25092.714,E2 -25092.714} C_VEL
LIN {X 0,Y 128.238,Z 766.188,A -85,B 0,C 180,E1 -25097.334,E2 -25097.334} C_VEL
LIN {X 0,Y 127.415,Z 767.575,A -85,B 0,C 180,E1 -25100.473,E2 -25100.473} C_VEL
LIN {X 0,Y 126.889,Z 768.561,A -85,B 0,C 180,E1 -25103.637,E2 -25103.637} C_VEL
LIN {X 0,Y 126.586,Z 769.167,A -85,B 0,C 180,E1 -25106.815,E2 -25106.815} C_VEL
LIN {X 0,Y 126.505,Z 769.393,A -85,B 0,C 180,E1 -25109.997,E2 -25109.997} C_VEL
LIN {X 0,Y 126.585,Z 769.198,A -85,B 0,C 180,E1 -25113.18,E2 -25113.18} C_VEL
LIN {X 0,Y 126.888,Z 768.613,A -85,B 0,C 180,E1 -25116.357,E2 -25116.357} C_VEL
LIN {X 0,Y 128.234,Z 766.293,A -85,B 0,C 180,E1 -25122.661,E2 -25122.661} C_VEL
LIN {X 0,Y 130.088,Z 763.421,A -85,B 0,C 180,E1 -25127.283,E2 -25127.283} C_VEL
LIN {X 0,Y 132.685,Z 759.524,A -85,B 0,C 180,E1 -25131.76,E2 -25131.76} C_VEL
LIN {X 0,Y 135.929,Z 754.503,A -85,B 0,C 180,E1 -25136.068,E2 -25136.068} C_VEL
LIN {X 0,Y 139.981,Z 748.168,A -85,B 0,C 180,E1 -25140.134,E2 -25140.134} C_VEL
LIN {X 0,Y 144.487,Z 740.234,A -85,B 0,C 180,E1 -25144.017,E2 -25144.017} C_VEL
LIN {X 0,Y 149.53,Z 730.395,A -85,B 0,C 180,E1 -25147.659,E2 -25147.659} C_VEL
LIN {X 0,Y 153.731,Z 721.208,A -85,B 0,C 180,E1 -25150.218,E2 -25150.218} C_VEL
LIN {X 0,Y 158.274,Z 709.78,A -85,B 0,C 180,E1 -25152.619,E2 -25152.619} C_VEL
LIN {X 0,Y 161.938,Z 698.542,A -85,B 0,C 180,E1 -25154.409,E2 -25154.409} C_VEL
LIN {X 0,Y 164.889,Z 687.106,A -85,B 0,C 180,E1 -25155.771,E2 -25155.771} C_VEL
LIN {X 0,Y 167.324,Z 673.83,A -85,B 0,C 180,E1 -25156.884,E2 -25156.884} C_VEL
LIN {X 0,Y 168.864,Z 660.385,A -85,B 0,C 180,E1 -25157.58,E2 -25157.58} C_VEL
LIN {X 0,Y 171.059,Z 629.379,A -85,B 0,C 180,E1 -25158.686,E2 -25158.686} C_VEL
LIN {X 0,Y 168.806,Z 623.972,A -85,B 0,C 180,E1 -25159.919,E2 -25159.919} C_VEL
LIN {X 0,Y 164.169,Z 615.309,A -85,B 0,C 180,E1 -25162.504,E2 -25162.504} C_VEL
LIN {X 0,Y 158.813,Z 606.318,A -85,B 0,C 180,E1 -25165.824,E2 -25165.824} C_VEL
LIN {X 0,Y 154.119,Z 599.22,A -85,B 0,C 180,E1 -25169.135,E2 -25169.135} C_VEL
LIN {X 0,Y 150.737,Z 594.609,A -85,B 0,C 180,E1 -25171.831,E2 -25171.831} C_VEL
LIN {X 0,Y 147.894,Z 590.678,A -85,B 0,C 180,E1 -25174.411,E2 -25174.411} C_VEL
LIN {X 0,Y 145.011,Z 587.168,A -85,B 0,C 180,E1 -25177.369,E2 -25177.369} C_VEL
LIN {X 0,Y 144.074,Z 585.662,A -85,B 0,C 180,E1 -25178.489,E2 -25178.489} C_VEL
LIN {X 0,Y 141.504,Z 583.189,A -85,B 0,C 180,E1 -25181.728,E2 -25181.728} C_VEL
LIN {X 0,Y 140.162,Z 580.432,A -85,B 0,C 180,E1 -25183.991,E2 -25183.991} C_VEL
LIN {X 0,Y 137.528,Z 578.607,A -85,B 0,C 180,E1 -25188.973,E2 -25188.973} C_VEL
LIN {X 0,Y 135.766,Z 574.829,A -85,B 0,C 180,E1 -25196.476,E2 -25196.476} C_VEL
LIN {X 0,Y 135.742,Z 574.452,A -85,B 0,C 180,E1 -25197.032,E2 -25197.032} C_VEL
LIN {X 0,Y 135.645,Z 574.403,A -85,B 0,C 180,E1 -25201.484,E2 -25201.484} C_VEL
LIN {X 0,Y 135.789,Z 574.844,A -85,B 0,C 180,E1 -25203.338,E2 -25203.338} C_VEL
LIN {X 0,Y 137.198,Z 578.191,A -85,B 0,C 180,E1 -25209.8,E2 -25209.8} C_VEL
LIN {X 0,Y 140.243,Z 580.695,A -85,B 0,C 180,E1 -25215.812,E2 -25215.812} C_VEL
LIN {X 0,Y 142.1,Z 583.972,A -85,B 0,C 180,E1 -25218.752,E2 -25218.752} C_VEL
LIN {X 0,Y 144.52,Z 586.238,A -85,B 0,C 180,E1 -25221.674,E2 -25221.674} C_VEL
LIN {X 0,Y 146.649,Z 589.438,A -85,B 0,C 180,E1 -25224.039,E2 -25224.039} C_VEL
LIN {X 0,Y 148.426,Z 591.353,A -85,B 0,C 180,E1 -25225.73,E2 -25225.73} C_VEL
LIN {X 0,Y 151.999,Z 596.329,A -85,B 0,C 180,E1 -25228.855,E2 -25228.855} C_VEL
LIN {X 0,Y 155.116,Z 600.781,A -85,B 0,C 180,E1 -25231.256,E2 -25231.256} C_VEL
LIN {X 0,Y 159.753,Z 609.329,A -85,B 0,C 180,E1 -25234.546,E2 -25234.546} C_VEL
LIN {X 0,Y 164.063,Z 618.412,A -85,B 0,C 180,E1 -25237.306,E2 -25237.306} C_VEL
LIN {X 0,Y 167.981,Z 627.982,A -85,B 0,C 180,E1 -25239.645,E2 -25239.645} C_VEL
LIN {X 0,Y 170.643,Z 635.432,A -85,B 0,C 180,E1 -25241.172,E2 -25241.172} C_VEL
LIN {X 0,Y 167.856,Z 673.321,A -85,B 0,C 180,E1 -25242.597,E2 -25242.597} C_VEL
LIN {X 0,Y 165.752,Z 686.862,A -85,B 0,C 180,E1 -25243.46,E2 -25243.46} C_VEL
LIN {X 0,Y 162.815,Z 699.121,A -85,B 0,C 180,E1 -25244.587,E2 -25244.587} C_VEL
LIN {X 0,Y 158.993,Z 711.786,A -85,B 0,C 180,E1 -25246.32,E2 -25246.32} C_VEL
LIN {X 0,Y 154.742,Z 723.043,A -85,B 0,C 180,E1 -25248.38,E2 -25248.38} C_VEL
LIN {X 0,Y 150.262,Z 733.184,A -85,B 0,C 180,E1 -25250.849,E2 -25250.849} C_VEL
LIN {X 0,Y 145.678,Z 742.33,A -85,B 0,C 180,E1 -25253.777,E2 -25253.777} C_VEL
LIN {X 0,Y 140.731,Z 751.385,A -85,B 0,C 180,E1 -25257.619,E2 -25257.619} C_VEL
LIN {X 0,Y 136.674,Z 758.431,A -85,B 0,C 180,E1 -25261.601,E2 -25261.601} C_VEL
LIN {X 0,Y 133.55,Z 763.275,A -85,B 0,C 180,E1 -25265.106,E2 -25265.106} C_VEL
LIN {X 0,Y 130.58,Z 767.99,A -85,B 0,C 180,E1 -25269.525,E2 -25269.525} C_VEL
LIN {X 0,Y 128.447,Z 771.601,A -85,B 0,C 180,E1 -25274.126,E2 -25274.126} C_VEL
LIN {X 0,Y 127.23,Z 773.869,A -85,B 0,C 180,E1 -25278.178,E2 -25278.178} C_VEL
LIN {X 0,Y 126.411,Z 775.86,A -85,B 0,C 180,E1 -25283.619,E2 -25283.619} C_VEL
LIN {X 0,Y 126.303,Z 776.471,A -85,B 0,C 180,E1 -25286.813,E2 -25286.813} C_VEL
LIN {X 0,Y 126.419,Z 776.686,A -85,B 0,C 180,E1 -25290.003,E2 -25290.003} C_VEL
LIN {X 0,Y 126.474,Z 776.55,A -85,B 0,C 180,E1 -25291.938,E2 -25291.938} C_VEL
LIN {X 0,Y 126.308,Z 776.373,A -85,B 0,C 180,E1 -25293.716,E2 -25293.716} C_VEL
LIN {X 0,Y 124.875,Z 775.594,A -85,B 0,C 180,E1 -25297.244,E2 -25297.244} C_VEL
LIN {X 0,Y 122.645,Z 773.562,A -85,B 0,C 180,E1 -25302.594,E2 -25302.594} C_VEL
LIN {X 0,Y 122.775,Z 772.159,A -85,B 0,C 180,E1 -25305.286,E2 -25305.286} C_VEL
LIN {X 0,Y 123.154,Z 771.603,A -85,B 0,C 180,E1 -25306.161,E2 -25306.161} C_VEL
LIN {X 0,Y 126.187,Z 768.69,A -85,B 0,C 180,E1 -25310.374,E2 -25310.374} C_VEL
LIN {X 0,Y 129.557,Z 773.391,A -85,B 0,C 180,E1 -25315.723,E2 -25315.723} C_VEL
LIN {X 0,Y 132.075,Z 775.709,A -85,B 0,C 180,E1 -25318.617,E2 -25318.617} C_VEL
LIN {X 0,Y 138.738,Z 779.181,A -85,B 0,C 180,E1 -25323.867,E2 -25323.867} C_VEL
LIN {X 0,Y 142.683,Z 780.473,A -85,B 0,C 180,E1 -25326.236,E2 -25326.236} C_VEL
LIN {X 0,Y 151.618,Z 781.852,A -85,B 0,C 180,E1 -25330.465,E2 -25330.465} C_VEL
LIN {X 0,Y 156.525,Z 782.075,A -85,B 0,C 180,E1 -25332.341,E2 -25332.341} C_VEL
LIN {X 0,Y 167.161,Z 781.317,A -85,B 0,C 180,E1 -25335.624,E2 -25335.624} C_VEL
LIN {X 0,Y 163.579,Z 781.651,A -85,B 0,C 180,E1 -25336.921,E2 -25336.921} C_VEL
LIN {X 0,Y 158.864,Z 781.866,A -85,B 0,C 180,E1 -25338.426,E2 -25338.426} C_VEL
LIN {X 0,Y 149.023,Z 781.188,A -85,B 0,C 180,E1 -25342.187,E2 -25342.187} C_VEL
LIN {X 0,Y 144.563,Z 780.294,A -85,B 0,C 180,E1 -25344.311,E2 -25344.311} C_VEL
LIN {X 0,Y 136.811,Z 777.379,A -85,B 0,C 180,E1 -25349.089,E2 -25349.089} C_VEL
LIN {X 0,Y 132.002,Z 774.182,A -85,B 0,C 180,E1 -25353.092,E2 -25353.092} C_VEL
LIN {X 0,Y 128.273,Z 770.129,A -85,B 0,C 180,E1 -25357.448,E2 -25357.448} C_VEL
LIN {X 0,Y 126.072,Z 765.962,A -85,B 0,C 180,E1 -25361.392,E2 -25361.392} C_VEL
LIN {X 0,Y 124.408,Z 759.089,A -85,B 0,C 180,E1 -25366.94,E2 -25366.94} C_VEL
LIN {X 0,Y 124.116,Z 751.658,A -85,B 0,C 180,E1 -25371.862,E2 -25371.862} C_VEL
LIN {X 0,Y 124.373,Z 743.986,A -85,B 0,C 180,E1 -25375.95,E2 -25375.95} C_VEL
LIN {X 0,Y 124.603,Z 736.178,A -85,B 0,C 180,E1 -25379.192,E2 -25379.192} C_VEL
LIN {X 0,Y 124.72,Z 727.556,A -85,B 0,C 180,E1 -25382.018,E2 -25382.018} C_VEL
LIN {X 0,Y 124.882,Z 718.451,A -85,B 0,C 180,E1 -25384.438,E2 -25384.438} C_VEL
LIN {X 0,Y 125.111,Z 706.82,A -85,B 0,C 180,E1 -25386.856,E2 -25386.856} C_VEL
LIN {X 0,Y 125.193,Z 696.736,A -85,B 0,C 180,E1 -25388.373,E2 -25388.373} C_VEL
LIN {X 0,Y 125.276,Z 678.909,A -85,B 0,C 180,E1 -25390.71,E2 -25390.71} C_VEL
LIN {X 0,Y 125.023,Z 675.95,A -85,B 0,C 180,E1 -25391.552,E2 -25391.552} C_VEL
LIN {X 0,Y 124.997,Z 674.865,A -85,B 0,C 180,E1 -25392.275,E2 -25392.275} C_VEL
LIN {X 0,Y 125.4,Z 674.683,A -85,B 0,C 180,E1 -25393.161,E2 -25393.161} C_VEL
LIN {X 0,Y 126.25,Z 673.152,A -85,B 0,C 180,E1 -25394.096,E2 -25394.096} C_VEL
LIN {X 0,Y 127.643,Z 669.484,A -85,B 0,C 180,E1 -25395.161,E2 -25395.161} C_VEL
LIN {X 0,Y 130.031,Z 660.467,A -85,B 0,C 180,E1 -25396.708,E2 -25396.708} C_VEL
LIN {X 0,Y 132.09,Z 651.464,A -85,B 0,C 180,E1 -25397.988,E2 -25397.988} C_VEL
LIN {X 0,Y 133.508,Z 649.625,A -85,B 0,C 180,E1 -25399.508,E2 -25399.508} C_VEL
LIN {X 0,Y 134.922,Z 646.43,A -85,B 0,C 180,E1 -25400.685,E2 -25400.685} C_VEL
LIN {X 0,Y 136.692,Z 641.06,A -85,B 0,C 180,E1 -25401.852,E2 -25401.852} C_VEL
LIN {X 0,Y 139.058,Z 632.128,A -85,B 0,C 180,E1 -25403.053,E2 -25403.053} C_VEL
LIN {X 0,Y 142.162,Z 628.842,A -85,B 0,C 180,E1 -25405.484,E2 -25405.484} C_VEL
LIN {X 0,Y 146.249,Z 623.398,A -85,B 0,C 180,E1 -25408.135,E2 -25408.135} C_VEL
LIN {X 0,Y 149.322,Z 621.979,A -85,B 0,C 180,E1 -25410.152,E2 -25410.152} C_VEL
LIN {X 0,Y 153.416,Z 618.602,A -85,B 0,C 180,E1 -25412.42,E2 -25412.42} C_VEL
LIN {X 0,Y 155.465,Z 616.57,A -85,B 0,C 180,E1 -25413.433,E2 -25413.433} C_VEL
LIN {X 0,Y 158.217,Z 616.037,A -85,B 0,C 180,E1 -25414.884,E2 -25414.884} C_VEL
LIN {X 0,Y 163.686,Z 626.159,A -85,B 0,C 180,E1 -25418.275,E2 -25418.275} C_VEL
LIN {X 0,Y 166.112,Z 631.46,A -85,B 0,C 180,E1 -25419.686,E2 -25419.686} C_VEL
LIN {X 0,Y 163.848,Z 661.712,A -85,B 0,C 180,E1 -25420.777,E2 -25420.777} C_VEL
LIN {X 0,Y 162.267,Z 674.292,A -85,B 0,C 180,E1 -25421.43,E2 -25421.43} C_VEL
LIN {X 0,Y 159.843,Z 687.334,A -85,B 0,C 180,E1 -25422.566,E2 -25422.566} C_VEL
LIN {X 0,Y 156.483,Z 699.638,A -85,B 0,C 180,E1 -25424.059,E2 -25424.059} C_VEL
LIN {X 0,Y 152.651,Z 710.7,A -85,B 0,C 180,E1 -25425.862,E2 -25425.862} C_VEL
LIN {X 0,Y 148.481,Z 720.831,A -85,B 0,C 180,E1 -25428.04,E2 -25428.04} C_VEL
LIN {X 0,Y 144.056,Z 730.134,A -85,B 0,C 180,E1 -25430.635,E2 -25430.635} C_VEL
LIN {X 0,Y 139.753,Z 738.26,A -85,B 0,C 180,E1 -25433.574,E2 -25433.574} C_VEL
LIN {X 0,Y 134.762,Z 746.839,A -85,B 0,C 180,E1 -25437.684,E2 -25437.684} C_VEL
LIN {X 0,Y 130.349,Z 753.477,A -85,B 0,C 180,E1 -25441.848,E2 -25441.848} C_VEL
LIN {X 0,Y 127.237,Z 757.968,A -85,B 0,C 180,E1 -25445.524,E2 -25445.524} C_VEL
LIN {X 0,Y 124.201,Z 762.272,A -85,B 0,C 180,E1 -25450.15,E2 -25450.15} C_VEL
LIN {X 0,Y 122.574,Z 764.547,A -85,B 0,C 180,E1 -25453.338,E2 -25453.338} C_VEL
LIN {X 0,Y 121.331,Z 766.393,A -85,B 0,C 180,E1 -25456.6,E2 -25456.6} C_VEL
LIN {X 0,Y 120.43,Z 767.78,A -85,B 0,C 180,E1 -25459.914,E2 -25459.914} C_VEL
LIN {X 0,Y 119.841,Z 768.766,A -85,B 0,C 180,E1 -25463.262,E2 -25463.262} C_VEL
LIN {X 0,Y 119.499,Z 769.372,A -85,B 0,C 180,E1 -25466.625,E2 -25466.625} C_VEL
LIN {X 0,Y 119.419,Z 769.597,A -85,B 0,C 180,E1 -25469.997,E2 -25469.997} C_VEL
LIN {X 0,Y 119.498,Z 769.402,A -85,B 0,C 180,E1 -25473.369,E2 -25473.369} C_VEL
LIN {X 0,Y 119.84,Z 768.817,A -85,B 0,C 180,E1 -25476.733,E2 -25476.733} C_VEL
LIN {X 0,Y 121.327,Z 766.496,A -85,B 0,C 180,E1 -25483.394,E2 -25483.394} C_VEL
LIN {X 0,Y 123.309,Z 763.626,A -85,B 0,C 180,E1 -25488.266,E2 -25488.266} C_VEL
LIN {X 0,Y 126.097,Z 759.729,A -85,B 0,C 180,E1 -25492.96,E2 -25492.96} C_VEL
LIN {X 0,Y 129.587,Z 754.706,A -85,B 0,C 180,E1 -25497.448,E2 -25497.448} C_VEL
LIN {X 0,Y 133.877,Z 748.371,A -85,B 0,C 180,E1 -25501.662,E2 -25501.662} C_VEL
LIN {X 0,Y 138.383,Z 740.921,A -85,B 0,C 180,E1 -25505.447,E2 -25505.447} C_VEL
LIN {X 0,Y 143.047,Z 732.374,A -85,B 0,C 180,E1 -25508.783,E2 -25508.783} C_VEL
LIN {X 0,Y 147.883,Z 722.513,A -85,B 0,C 180,E1 -25511.705,E2 -25511.705} C_VEL
LIN {X 0,Y 152.597,Z 711.402,A -85,B 0,C 180,E1 -25514.151,E2 -25514.151} C_VEL
LIN {X 0,Y 156.408,Z 700.504,A -85,B 0,C 180,E1 -25515.963,E2 -25515.963} C_VEL
LIN {X 0,Y 159.741,Z 688.446,A -85,B 0,C 180,E1 -25517.467,E2 -25517.467} C_VEL
LIN {X 0,Y 162.321,Z 675.579,A -85,B 0,C 180,E1 -25518.605,E2 -25518.605} C_VEL
LIN {X 0,Y 163.98,Z 662.593,A -85,B 0,C 180,E1 -25519.324,E2 -25519.324} C_VEL
LIN {X 0,Y 166.302,Z 631.681,A -85,B 0,C 180,E1 -25520.446,E2 -25520.446} C_VEL
LIN {X 0,Y 163.535,Z 625.644,A -85,B 0,C 180,E1 -25522.064,E2 -25522.064} C_VEL
LIN {X 0,Y 157.589,Z 614.813,A -85,B 0,C 180,E1 -25525.806,E2 -25525.806} C_VEL
LIN {X 0,Y 152.933,Z 607.276,A -85,B 0,C 180,E1 -25529.157,E2 -25529.157} C_VEL
LIN {X 0,Y 148.625,Z 600.961,A -85,B 0,C 180,E1 -25532.736,E2 -25532.736} C_VEL
LIN {X 0,Y 145.733,Z 596.923,A -85,B 0,C 180,E1 -25535.52,E2 -25535.52} C_VEL
LIN {X 0,Y 143.007,Z 593.264,A -85,B 0,C 180,E1 -25538.556,E2 -25538.556} C_VEL
LIN {X 0,Y 142.212,Z 592.199,A -85,B 0,C 180,E1 -25539.547,E2 -25539.547} C_VEL
LIN {X 0,Y 139.622,Z 589.185,A -85,B 0,C 180,E1 -25543.176,E2 -25543.176} C_VEL
LIN {X 0,Y 138.659,Z 587.232,A -85,B 0,C 180,E1 -25544.944,E2 -25544.944} C_VEL
LIN {X 0,Y 136.092,Z 585.077,A -85,B 0,C 180,E1 -25550.451,E2 -25550.451} C_VEL
LIN {X 0,Y 134.808,Z 581.46,A -85,B 0,C 180,E1 -25557.759,E2 -25557.759} C_VEL
LIN {X 0,Y 134.857,Z 581.655,A -85,B 0,C 180,E1 -25562.613,E2 -25562.613} C_VEL
LIN {X 0,Y 135.587,Z 584.171,A -85,B 0,C 180,E1 -25567.445,E2 -25567.445} C_VEL
LIN {X 0,Y 138.238,Z 587,A -85,B 0,C 180,E1 -25573.974,E2 -25573.974} C_VEL
LIN {X 0,Y 138.887,Z 587.645,A -85,B 0,C 180,E1 -25575.124,E2 -25575.124} C_VEL
LIN {X 0,Y 140.837,Z 590.888,A -85,B 0,C 180,E1 -25578.314,E2 -25578.314} C_VEL
LIN {X 0,Y 142.807,Z 592.911,A -85,B 0,C 180,E1 -25580.827,E2 -25580.827} C_VEL
LIN {X 0,Y 145.28,Z 596.444,A -85,B 0,C 180,E1 -25583.663,E2 -25583.663} C_VEL
LIN {X 0,Y 146.519,Z 597.977,A -85,B 0,C 180,E1 -25584.911,E2 -25584.911} C_VEL
LIN {X 0,Y 149.836,Z 602.731,A -85,B 0,C 180,E1 -25587.972,E2 -25587.972} C_VEL
LIN {X 0,Y 152.331,Z 606.413,A -85,B 0,C 180,E1 -25590.019,E2 -25590.019} C_VEL
LIN {X 0,Y 156.594,Z 614.668,A -85,B 0,C 180,E1 -25593.279,E2 -25593.279} C_VEL
LIN {X 0,Y 160.419,Z 623.123,A -85,B 0,C 180,E1 -25595.927,E2 -25595.927} C_VEL
LIN {X 0,Y 164.062,Z 632.366,A -85,B 0,C 180,E1 -25598.278,E2 -25598.278} C_VEL
LIN {X 0,Y 165.825,Z 637.562,A -85,B 0,C 180,E1 -25599.386,E2 -25599.386} C_VEL
LIN {X 0,Y 163.802,Z 666.493,A -85,B 0,C 180,E1 -25600.472,E2 -25600.472} C_VEL
LIN {X 0,Y 162.259,Z 679.559,A -85,B 0,C 180,E1 -25601.133,E2 -25601.133} C_VEL
LIN {X 0,Y 159.739,Z 691.971,A -85,B 0,C 180,E1 -25602.063,E2 -25602.063} C_VEL
LIN {X 0,Y 156.763,Z 702.913,A -85,B 0,C 180,E1 -25603.241,E2 -25603.241} C_VEL
LIN {X 0,Y 152.779,Z 714.684,A -85,B 0,C 180,E1 -25604.991,E2 -25604.991} C_VEL
LIN {X 0,Y 147.934,Z 726.44,A -85,B 0,C 180,E1 -25607.395,E2 -25607.395} C_VEL
LIN {X 0,Y 142.835,Z 736.881,A -85,B 0,C 180,E1 -25610.238,E2 -25610.238} C_VEL
LIN {X 0,Y 138.205,Z 745.335,A -85,B 0,C 180,E1 -25613.312,E2 -25613.312} C_VEL
LIN {X 0,Y 133.321,Z 753.599,A -85,B 0,C 180,E1 -25617.297,E2 -25617.297} C_VEL
LIN {X 0,Y 129.081,Z 760.26,A -85,B 0,C 180,E1 -25621.552,E2 -25621.552} C_VEL
LIN {X 0,Y 124.919,Z 766.351,A -85,B 0,C 180,E1 -25626.811,E2 -25626.811} C_VEL
LIN {X 0,Y 122.247,Z 770.318,A -85,B 0,C 180,E1 -25631.57,E2 -25631.57} C_VEL
LIN {X 0,Y 120.524,Z 773.258,A -85,B 0,C 180,E1 -25636.515,E2 -25636.515} C_VEL
LIN {X 0,Y 119.784,Z 774.656,A -85,B 0,C 180,E1 -25639.865,E2 -25639.865} C_VEL
LIN {X 0,Y 119.219,Z 776.267,A -85,B 0,C 180,E1 -25646.623,E2 -25646.623} C_VEL
LIN {X 0,Y 119.33,Z 776.482,A -85,B 0,C 180,E1 -25650.003,E2 -25650.003} C_VEL
LIN {X 0,Y 119.5,Z 776.257,A -85,B 0,C 180,E1 -25653.374,E2 -25653.374} C_VEL
LIN {X 0,Y 119.915,Z 775.642,A -85,B 0,C 180,E1 -25656.734,E2 -25656.734} C_VEL
LIN {X 0,Y 121.765,Z 773.234,A -85,B 0,C 180,E1 -25663.351,E2 -25663.351} C_VEL
LIN {X 0,Y 123.154,Z 771.603,A -85,B 0,C 180,E1 -25666.161,E2 -25666.161} C_VEL
LIN {X 0,Y 123.575,Z 770.562,A -85,B 0,C 180,E1 -25667.985,E2 -25667.985} C_VEL
LIN {X 0,Y 122.84,Z 769.252,A -85,B 0,C 180,E1 -25671.113,E2 -25671.113} C_VEL
LIN {X 0,Y 122.255,Z 769.09,A -85,B 0,C 180,E1 -25673.646,E2 -25673.646} C_VEL
LIN {X 0,Y 122.574,Z 769.889,A -85,B 0,C 180,E1 -25675.639,E2 -25675.639} C_VEL
LIN {X 0,Y 122.818,Z 770.228,A -85,B 0,C 180,E1 -25676.066,E2 -25676.066} C_VEL
LIN {X 0,Y 126.165,Z 773.677,A -85,B 0,C 180,E1 -25680.092,E2 -25680.092} C_VEL
LIN {X 0,Y 129.318,Z 775.906,A -85,B 0,C 180,E1 -25682.923,E2 -25682.923} C_VEL
LIN {X 0,Y 137.119,Z 779.253,A -85,B 0,C 180,E1 -25687.959,E2 -25687.959} C_VEL
LIN {X 0,Y 141.543,Z 780.484,A -85,B 0,C 180,E1 -25690.205,E2 -25690.205} C_VEL
LIN {X 0,Y 151.351,Z 781.771,A -85,B 0,C 180,E1 -25694.152,E2 -25694.152} C_VEL
LIN {X 0,Y 154.998,Z 781.925,A -85,B 0,C 180,E1 -25695.336,E2 -25695.336} C_VEL
LIN {X 0,Y 155.609,Z 781.934,A -85,B 0,C 180,E1 -25696.027,E2 -25696.027} C_VEL
LIN {X 0,Y 148.406,Z 781.4,A -85,B 0,C 180,E1 -25698.472,E2 -25698.472} C_VEL
LIN {X 0,Y 138.913,Z 779.275,A -85,B 0,C 180,E1 -25702.619,E2 -25702.619} C_VEL
LIN {X 0,Y 134.736,Z 777.791,A -85,B 0,C 180,E1 -25704.986,E2 -25704.986} C_VEL
LIN {X 0,Y 127.487,Z 773.483,A -85,B 0,C 180,E1 -25710.255,E2 -25710.255} C_VEL
LIN {X 0,Y 123.293,Z 769.308,A -85,B 0,C 180,E1 -25714.69,E2 -25714.69} C_VEL
LIN {X 0,Y 119.866,Z 763.268,A -85,B 0,C 180,E1 -25720.39,E2 -25720.39} C_VEL
LIN {X 0,Y 118.184,Z 755.829,A -85,B 0,C 180,E1 -25726.239,E2 -25726.239} C_VEL
LIN {X 0,Y 117.933,Z 749.369,A -85,B 0,C 180,E1 -25730.568,E2 -25730.568} C_VEL
LIN {X 0,Y 118.158,Z 743.119,A -85,B 0,C 180,E1 -25734.025,E2 -25734.025} C_VEL
LIN {X 0,Y 118.329,Z 735.42,A -85,B 0,C 180,E1 -25737.447,E2 -25737.447} C_VEL
LIN {X 0,Y 118.369,Z 727.008,A -85,B 0,C 180,E1 -25740.425,E2 -25740.425} C_VEL
LIN {X 0,Y 118.434,Z 717.94,A -85,B 0,C 180,E1 -25742.977,E2 -25742.977} C_VEL
LIN {X 0,Y 118.615,Z 706.234,A -85,B 0,C 180,E1 -25745.525,E2 -25745.525} C_VEL
LIN {X 0,Y 118.543,Z 695.433,A -85,B 0,C 180,E1 -25747.345,E2 -25747.345} C_VEL
LIN {X 0,Y 118.196,Z 693.034,A -85,B 0,C 180,E1 -25748.334,E2 -25748.334} C_VEL
LIN {X 0,Y 118.112,Z 692.762,A -85,B 0,C 180,E1 -25748.986,E2 -25748.986} C_VEL
LIN {X 0,Y 118.652,Z 692.334,A -85,B 0,C 180,E1 -25750.236,E2 -25750.236} C_VEL
LIN {X 0,Y 119.999,Z 690.081,A -85,B 0,C 180,E1 -25751.484,E2 -25751.484} C_VEL
LIN {X 0,Y 122.037,Z 685.918,A -85,B 0,C 180,E1 -25752.747,E2 -25752.747} C_VEL
LIN {X 0,Y 123.87,Z 681.629,A -85,B 0,C 180,E1 -25753.744,E2 -25753.744} C_VEL
LIN {X 0,Y 125.303,Z 680.006,A -85,B 0,C 180,E1 -25755.451,E2 -25755.451} C_VEL
LIN {X 0,Y 127.17,Z 676.526,A -85,B 0,C 180,E1 -25756.97,E2 -25756.97} C_VEL
LIN {X 0,Y 129.147,Z 671.68,A -85,B 0,C 180,E1 -25758.132,E2 -25758.132} C_VEL
LIN {X 0,Y 131.694,Z 663.173,A -85,B 0,C 180,E1 -25759.484,E2 -25759.484} C_VEL
LIN {X 0,Y 133.271,Z 656.813,A -85,B 0,C 180,E1 -25760.348,E2 -25760.348} C_VEL
LIN {X 0,Y 135.149,Z 653.767,A -85,B 0,C 180,E1 -25761.996,E2 -25761.996} C_VEL
LIN {X 0,Y 137.144,Z 649.094,A -85,B 0,C 180,E1 -25763.394,E2 -25763.394} C_VEL
LIN {X 0,Y 139.299,Z 642.55,A -85,B 0,C 180,E1 -25764.596,E2 -25764.596} C_VEL
LIN {X 0,Y 140.795,Z 637.375,A -85,B 0,C 180,E1 -25765.304,E2 -25765.304} C_VEL
LIN {X 0,Y 144.529,Z 633.126,A -85,B 0,C 180,E1 -25767.858,E2 -25767.858} C_VEL
LIN {X 0,Y 146.907,Z 630.089,A -85,B 0,C 180,E1 -25769.282,E2 -25769.282} C_VEL
LIN {X 0,Y 150.759,Z 628.004,A -85,B 0,C 180,E1 -25771.631,E2 -25771.631} C_VEL
LIN {X 0,Y 155.702,Z 623.765,A -85,B 0,C 180,E1 -25774.153,E2 -25774.153} C_VEL
LIN {X 0,Y 156.223,Z 623.478,A -85,B 0,C 180,E1 -25774.413,E2 -25774.413} C_VEL
LIN {X 0,Y 160.719,Z 632.352,A -85,B 0,C 180,E1 -25777.354,E2 -25777.354} C_VEL
LIN {X 0,Y 161.511,Z 634.047,A -85,B 0,C 180,E1 -25777.844,E2 -25777.844} C_VEL
LIN {X 0,Y 158.937,Z 665.453,A -85,B 0,C 180,E1 -25778.977,E2 -25778.977} C_VEL
LIN {X 0,Y 156.925,Z 678.856,A -85,B 0,C 180,E1 -25779.829,E2 -25779.829} C_VEL
LIN {X 0,Y 153.975,Z 692.069,A -85,B 0,C 180,E1 -25781.136,E2 -25781.136} C_VEL
LIN {X 0,Y 150.516,Z 703.334,A -85,B 0,C 180,E1 -25782.655,E2 -25782.655} C_VEL
LIN {X 0,Y 145.989,Z 714.954,A -85,B 0,C 180,E1 -25784.756,E2 -25784.756} C_VEL
LIN {X 0,Y 141.186,Z 725.393,A -85,B 0,C 180,E1 -25787.292,E2 -25787.292} C_VEL
LIN {X 0,Y 136.685,Z 733.917,A -85,B 0,C 180,E1 -25790.002,E2 -25790.002} C_VEL
LIN {X 0,Y 131.975,Z 742.006,A -85,B 0,C 180,E1 -25793.347,E2 -25793.347} C_VEL
LIN {X 0,Y 127.181,Z 749.436,A -85,B 0,C 180,E1 -25797.396,E2 -25797.396} C_VEL
LIN {X 0,Y 122.012,Z 756.487,A -85,B 0,C 180,E1 -25802.558,E2 -25802.558} C_VEL
LIN {X 0,Y 118.549,Z 761.172,A -85,B 0,C 180,E1 -25807.332,E2 -25807.332} C_VEL
LIN {X 0,Y 115.796,Z 764.752,A -85,B 0,C 180,E1 -25812.331,E2 -25812.331} C_VEL
LIN {X 0,Y 114.429,Z 766.599,A -85,B 0,C 180,E1 -25815.775,E2 -25815.775} C_VEL
LIN {X 0,Y 113.433,Z 767.985,A -85,B 0,C 180,E1 -25819.285,E2 -25819.285} C_VEL
LIN {X 0,Y 112.791,Z 768.971,A -85,B 0,C 180,E1 -25822.838,E2 -25822.838} C_VEL
LIN {X 0,Y 112.425,Z 769.576,A -85,B 0,C 180,E1 -25826.413,E2 -25826.413} C_VEL
LIN {X 0,Y 112.335,Z 769.801,A -85,B 0,C 180,E1 -25829.997,E2 -25829.997} C_VEL
LIN {X 0,Y 112.424,Z 769.606,A -85,B 0,C 180,E1 -25833.581,E2 -25833.581} C_VEL
LIN {X 0,Y 112.789,Z 769.022,A -85,B 0,C 180,E1 -25837.156,E2 -25837.156} C_VEL
LIN {X 0,Y 114.424,Z 766.701,A -85,B 0,C 180,E1 -25844.219,E2 -25844.219} C_VEL
LIN {X 0,Y 116.577,Z 763.83,A -85,B 0,C 180,E1 -25849.361,E2 -25849.361} C_VEL
LIN {X 0,Y 119.57,Z 759.933,A -85,B 0,C 180,E1 -25854.292,E2 -25854.292} C_VEL
LIN {X 0,Y 123.332,Z 754.909,A -85,B 0,C 180,E1 -25858.968,E2 -25858.968} C_VEL
LIN {X 0,Y 127.881,Z 748.574,A -85,B 0,C 180,E1 -25863.334,E2 -25863.334} C_VEL
LIN {X 0,Y 132.36,Z 741.627,A -85,B 0,C 180,E1 -25867.001,E2 -25867.001} C_VEL
LIN {X 0,Y 137.575,Z 732.577,A -85,B 0,C 180,E1 -25870.639,E2 -25870.639} C_VEL
LIN {X 0,Y 142.676,Z 722.714,A -85,B 0,C 180,E1 -25873.596,E2 -25873.596} C_VEL
LIN {X 0,Y 147.597,Z 711.602,A -85,B 0,C 180,E1 -25876.067,E2 -25876.067} C_VEL
LIN {X 0,Y 151.566,Z 700.703,A -85,B 0,C 180,E1 -25877.89,E2 -25877.89} C_VEL
LIN {X 0,Y 155.046,Z 688.643,A -85,B 0,C 180,E1 -25879.394,E2 -25879.394} C_VEL
LIN {X 0,Y 157.673,Z 676.079,A -85,B 0,C 180,E1 -25880.517,E2 -25880.517} C_VEL
LIN {X 0,Y 159.443,Z 662.879,A -85,B 0,C 180,E1 -25881.251,E2 -25881.251} C_VEL
LIN {X 0,Y 161.692,Z 634.178,A -85,B 0,C 180,E1 -25882.302,E2 -25882.302} C_VEL
LIN {X 0,Y 157.067,Z 624.931,A -85,B 0,C 180,E1 -25885.281,E2 -25885.281} C_VEL
LIN {X 0,Y 152.506,Z 616.712,A -85,B 0,C 180,E1 -25888.579,E2 -25888.579} C_VEL
LIN {X 0,Y 148.605,Z 610.489,A -85,B 0,C 180,E1 -25891.775,E2 -25891.775} C_VEL
LIN {X 0,Y 146.048,Z 606.65,A -85,B 0,C 180,E1 -25894.145,E2 -25894.145} C_VEL
LIN {X 0,Y 143.837,Z 603.372,A -85,B 0,C 180,E1 -25896.443,E2 -25896.443} C_VEL
LIN {X 0,Y 141.059,Z 599.405,A -85,B 0,C 180,E1 -25899.778,E2 -25899.778} C_VEL
LIN {X 0,Y 138.019,Z 595.558,A -85,B 0,C 180,E1 -25904.305,E2 -25904.305} C_VEL
LIN {X 0,Y 137.298,Z 594.068,A -85,B 0,C 180,E1 -25905.739,E2 -25905.739} C_VEL
LIN {X 0,Y 134.66,Z 591.351,A -85,B 0,C 180,E1 -25912.314,E2 -25912.314} C_VEL
LIN {X 0,Y 133.931,Z 588.607,A -85,B 0,C 180,E1 -25917.744,E2 -25917.744} C_VEL
LIN {X 0,Y 133.936,Z 588.558,A -85,B 0,C 180,E1 -25921.879,E2 -25921.879} C_VEL
LIN {X 0,Y 135.913,Z 593.039,A -85,B 0,C 180,E1 -25931.076,E2 -25931.076} C_VEL
LIN {X 0,Y 137.473,Z 594.333,A -85,B 0,C 180,E1 -25934.243,E2 -25934.243} C_VEL
LIN {X 0,Y 139.516,Z 597.783,A -85,B 0,C 180,E1 -25937.782,E2 -25937.782} C_VEL
LIN {X 0,Y 141.106,Z 599.52,A -85,B 0,C 180,E1 -25939.929,E2 -25939.929} C_VEL
LIN {X 0,Y 143.817,Z 603.328,A -85,B 0,C 180,E1 -25943.172,E2 -25943.172} C_VEL
LIN {X 0,Y 147.453,Z 608.735,A -85,B 0,C 180,E1 -25946.828,E2 -25946.828} C_VEL
LIN {X 0,Y 150.061,Z 612.871,A -85,B 0,C 180,E1 -25949.12,E2 -25949.12} C_VEL
LIN {X 0,Y 154.207,Z 621.468,A -85,B 0,C 180,E1 -25952.491,E2 -25952.491} C_VEL
LIN {X 0,Y 158.353,Z 631.474,A -85,B 0,C 180,E1 -25955.53,E2 -25955.53} C_VEL
LIN {X 0,Y 161.315,Z 640.076,A -85,B 0,C 180,E1 -25957.585,E2 -25957.585} C_VEL
LIN {X 0,Y 158.586,Z 672.958,A -85,B 0,C 180,E1 -25958.818,E2 -25958.818} C_VEL
LIN {X 0,Y 156.363,Z 686.421,A -85,B 0,C 180,E1 -25959.688,E2 -25959.688} C_VEL
LIN {X 0,Y 153.185,Z 698.724,A -85,B 0,C 180,E1 -25960.803,E2 -25960.803} C_VEL
LIN {X 0,Y 149.044,Z 711.386,A -85,B 0,C 180,E1 -25962.546,E2 -25962.546} C_VEL
LIN {X 0,Y 144.424,Z 722.641,A -85,B 0,C 180,E1 -25964.632,E2 -25964.632} C_VEL
LIN {X 0,Y 139.528,Z 732.78,A -85,B 0,C 180,E1 -25967.161,E2 -25967.161} C_VEL
LIN {X 0,Y 134.467,Z 741.925,A -85,B 0,C 180,E1 -25970.193,E2 -25970.193} C_VEL
LIN {X 0,Y 128.977,Z 750.841,A -85,B 0,C 180,E1 -25974.146,E2 -25974.146} C_VEL
LIN {X 0,Y 124.325,Z 757.985,A -85,B 0,C 180,E1 -25978.443,E2 -25978.443} C_VEL
LIN {X 0,Y 120.759,Z 762.867,A -85,B 0,C 180,E1 -25982.255,E2 -25982.255} C_VEL
LIN {X 0,Y 117.346,Z 767.581,A -85,B 0,C 180,E1 -25987.093,E2 -25987.093} C_VEL
LIN {X 0,Y 114.774,Z 771.19,A -85,B 0,C 180,E1 -25992.175,E2 -25992.175} C_VEL
LIN {X 0,Y 113.615,Z 773.054,A -85,B 0,C 180,E1 -25995.678,E2 -25995.678} C_VEL
LIN {X 0,Y 112.776,Z 774.451,A -85,B 0,C 180,E1 -25999.228,E2 -25999.228} C_VEL
LIN {X 0,Y 112.127,Z 776.062,A -85,B 0,C 180,E1 -26006.41,E2 -26006.41} C_VEL
LIN {X 0,Y 112.248,Z 776.277,A -85,B 0,C 180,E1 -26010.003,E2 -26010.003} C_VEL
LIN {X 0,Y 112.426,Z 776.053,A -85,B 0,C 180,E1 -26013.587,E2 -26013.587} C_VEL
LIN {X 0,Y 113.666,Z 774.433,A -85,B 0,C 180,E1 -26020.693,E2 -26020.693} C_VEL
LIN {X 0,Y 114.875,Z 773.029,A -85,B 0,C 180,E1 -26024.168,E2 -26024.168} C_VEL
LIN {X 0,Y 117.641,Z 770.1,A -85,B 0,C 180,E1 -26029.185,E2 -26029.185} C_VEL
LIN {X 0,Y 120.697,Z 767.386,A -85,B 0,C 180,E1 -26032.807,E2 -26032.807} C_VEL
LIN {X 0,Y 122.818,Z 770.228,A -85,B 0,C 180,E1 -26036.066,E2 -26036.066} C_VEL
LIN {X 0,Y 124.099,Z 772.172,A -85,B 0,C 180,E1 -26038.596,E2 -26038.596} C_VEL
LIN {X 0,Y 127.415,Z 775.877,A -85,B 0,C 180,E1 -26046.4,E2 -26046.4} C_VEL
LIN {X 0,Y 129.873,Z 777.046,A -85,B 0,C 180,E1 -26048.717,E2 -26048.717} C_VEL
LIN {X 0,Y 130.964,Z 777.499,A -85,B 0,C 180,E1 -26049.403,E2 -26049.403} C_VEL
LIN {X 0,Y 141.162,Z 780.447,A -85,B 0,C 180,E1 -26054.191,E2 -26054.191} C_VEL
LIN {X 0,Y 143.229,Z 780.756,A -85,B 0,C 180,E1 -26054.965,E2 -26054.965} C_VEL
LIN {X 0,Y 144.29,Z 780.88,A -85,B 0,C 180,E1 -26056.202,E2 -26056.202} C_VEL
LIN {X 0,Y 138.141,Z 779.541,A -85,B 0,C 180,E1 -26058.595,E2 -26058.595} C_VEL
LIN {X 0,Y 133.419,Z 778.075,A -85,B 0,C 180,E1 -26060.794,E2 -26060.794} C_VEL
LIN {X 0,Y 125.188,Z 773.971,A -85,B 0,C 180,E1 -26065.848,E2 -26065.848} C_VEL
LIN {X 0,Y 120.102,Z 769.927,A -85,B 0,C 180,E1 -26070.172,E2 -26070.172} C_VEL
LIN {X 0,Y 116.164,Z 765.061,A -85,B 0,C 180,E1 -26074.944,E2 -26074.944} C_VEL
LIN {X 0,Y 113.313,Z 758.631,A -85,B 0,C 180,E1 -26080.575,E2 -26080.575} C_VEL
LIN {X 0,Y 112.131,Z 752.257,A -85,B 0,C 180,E1 -26085.481,E2 -26085.481} C_VEL
LIN {X 0,Y 111.974,Z 743.773,A -85,B 0,C 180,E1 -26090.972,E2 -26090.972} C_VEL
LIN {X 0,Y 112.164,Z 736.685,A -85,B 0,C 180,E1 -26094.607,E2 -26094.607} C_VEL
LIN {X 0,Y 112.159,Z 728.721,A -85,B 0,C 180,E1 -26097.756,E2 -26097.756} C_VEL
LIN {X 0,Y 112.175,Z 718.778,A -85,B 0,C 180,E1 -26100.898,E2 -26100.898} C_VEL
LIN {X 0,Y 112.145,Z 707.259,A -85,B 0,C 180,E1 -26103.818,E2 -26103.818} C_VEL
LIN {X 0,Y 111.682,Z 705.572,A -85,B 0,C 180,E1 -26104.851,E2 -26104.851} C_VEL
LIN {X 0,Y 111.545,Z 705.405,A -85,B 0,C 180,E1 -26105.423,E2 -26105.423} C_VEL
LIN {X 0,Y 112.113,Z 704.898,A -85,B 0,C 180,E1 -26107.203,E2 -26107.203} C_VEL
LIN {X 0,Y 113.818,Z 702.366,A -85,B 0,C 180,E1 -26108.882,E2 -26108.882} C_VEL
LIN {X 0,Y 115.064,Z 700.273,A -85,B 0,C 180,E1 -26109.671,E2 -26109.671} C_VEL
LIN {X 0,Y 115.899,Z 699.102,A -85,B 0,C 180,E1 -26110.482,E2 -26110.482} C_VEL
LIN {X 0,Y 117.01,Z 698.019,A -85,B 0,C 180,E1 -26112.136,E2 -26112.136} C_VEL
LIN {X 0,Y 119.45,Z 694.508,A -85,B 0,C 180,E1 -26114.117,E2 -26114.117} C_VEL
LIN {X 0,Y 121.996,Z 689.97,A -85,B 0,C 180,E1 -26115.523,E2 -26115.523} C_VEL
LIN {X 0,Y 123.116,Z 687.756,A -85,B 0,C 180,E1 -26115.98,E2 -26115.98} C_VEL
LIN {X 0,Y 126.177,Z 683.532,A -85,B 0,C 180,E1 -26118.492,E2 -26118.492} C_VEL
LIN {X 0,Y 128.806,Z 678.862,A -85,B 0,C 180,E1 -26120.043,E2 -26120.043} C_VEL
LIN {X 0,Y 132.281,Z 670.187,A -85,B 0,C 180,E1 -26121.629,E2 -26121.629} C_VEL
LIN {X 0,Y 134.896,Z 661.485,A -85,B 0,C 180,E1 -26122.799,E2 -26122.799} C_VEL
LIN {X 0,Y 137.456,Z 656.943,A -85,B 0,C 180,E1 -26124.685,E2 -26124.685} C_VEL
LIN {X 0,Y 140.241,Z 650.107,A -85,B 0,C 180,E1 -26126.308,E2 -26126.308} C_VEL
LIN {X 0,Y 142.809,Z 642.355,A -85,B 0,C 180,E1 -26127.518,E2 -26127.518} C_VEL
LIN {X 0,Y 147.767,Z 636.648,A -85,B 0,C 180,E1 -26130.502,E2 -26130.502} C_VEL
LIN {X 0,Y 152.37,Z 633.884,A -85,B 0,C 180,E1 -26133.113,E2 -26133.113} C_VEL
LIN {X 0,Y 154.074,Z 632.561,A -85,B 0,C 180,E1 -26133.972,E2 -26133.972} C_VEL
LIN {X 0,Y 155.15,Z 632.862,A -85,B 0,C 180,E1 -26134.586,E2 -26134.586} C_VEL
LIN {X 0,Y 157.054,Z 636.953,A -85,B 0,C 180,E1 -26135.905,E2 -26135.905} C_VEL
LIN {X 0,Y 154.616,Z 665.361,A -85,B 0,C 180,E1 -26136.923,E2 -26136.923} C_VEL
LIN {X 0,Y 152.591,Z 678.563,A -85,B 0,C 180,E1 -26137.747,E2 -26137.747} C_VEL
LIN {X 0,Y 149.695,Z 691.154,A -85,B 0,C 180,E1 -26138.956,E2 -26138.956} C_VEL
LIN {X 0,Y 146.377,Z 701.82,A -85,B 0,C 180,E1 -26140.338,E2 -26140.338} C_VEL
LIN {X 0,Y 142.253,Z 712.54,A -85,B 0,C 180,E1 -26142.174,E2 -26142.174} C_VEL
LIN {X 0,Y 137.145,Z 723.469,A -85,B 0,C 180,E1 -26144.679,E2 -26144.679} C_VEL
LIN {X 0,Y 132.341,Z 732.35,A -85,B 0,C 180,E1 -26147.38,E2 -26147.38} C_VEL
LIN {X 0,Y 126.82,Z 741.479,A -85,B 0,C 180,E1 -26151.086,E2 -26151.086} C_VEL
LIN {X 0,Y 122.099,Z 748.479,A -85,B 0,C 180,E1 -26154.855,E2 -26154.855} C_VEL
LIN {X 0,Y 117.258,Z 754.885,A -85,B 0,C 180,E1 -26159.369,E2 -26159.369} C_VEL
LIN {X 0,Y 113.191,Z 759.964,A -85,B 0,C 180,E1 -26164.235,E2 -26164.235} C_VEL
LIN {X 0,Y 109.93,Z 763.902,A -85,B 0,C 180,E1 -26169.41,E2 -26169.41} C_VEL
LIN {X 0,Y 107.564,Z 766.804,A -85,B 0,C 180,E1 -26174.847,E2 -26174.847} C_VEL
LIN {X 0,Y 105.746,Z 769.176,A -85,B 0,C 180,E1 -26182.358,E2 -26182.358} C_VEL
LIN {X 0,Y 105.344,Z 769.781,A -85,B 0,C 180,E1 -26186.171,E2 -26186.171} C_VEL
LIN {X 0,Y 105.238,Z 770.006,A -85,B 0,C 180,E1 -26189.997,E2 -26189.997} C_VEL
LIN {X 0,Y 105.343,Z 769.811,A -85,B 0,C 180,E1 -26193.822,E2 -26193.822} C_VEL
LIN {X 0,Y 105.744,Z 769.226,A -85,B 0,C 180,E1 -26197.635,E2 -26197.635} C_VEL
LIN {X 0,Y 107.559,Z 766.905,A -85,B 0,C 180,E1 -26205.148,E2 -26205.148} C_VEL
LIN {X 0,Y 109.9,Z 764.034,A -85,B 0,C 180,E1 -26210.589,E2 -26210.589} C_VEL
LIN {X 0,Y 113.116,Z 760.137,A -85,B 0,C 180,E1 -26215.776,E2 -26215.776} C_VEL
LIN {X 0,Y 117.176,Z 755.112,A -85,B 0,C 180,E1 -26220.648,E2 -26220.648} C_VEL
LIN {X 0,Y 122.005,Z 748.777,A -85,B 0,C 180,E1 -26225.169,E2 -26225.169} C_VEL
LIN {X 0,Y 127.55,Z 740.56,A -85,B 0,C 180,E1 -26229.52,E2 -26229.52} C_VEL
LIN {X 0,Y 133.311,Z 731,A -85,B 0,C 180,E1 -26233.259,E2 -26233.259} C_VEL
LIN {X 0,Y 138.75,Z 720.639,A -85,B 0,C 180,E1 -26236.199,E2 -26236.199} C_VEL
LIN {X 0,Y 143.943,Z 708.957,A -85,B 0,C 180,E1 -26238.645,E2 -26238.645} C_VEL
LIN {X 0,Y 148.062,Z 697.278,A -85,B 0,C 180,E1 -26240.469,E2 -26240.469} C_VEL
LIN {X 0,Y 151.452,Z 685.118,A -85,B 0,C 180,E1 -26241.806,E2 -26241.806} C_VEL
LIN {X 0,Y 153.972,Z 671.957,A -85,B 0,C 180,E1 -26242.855,E2 -26242.855} C_VEL
LIN {X 0,Y 155.559,Z 658.019,A -85,B 0,C 180,E1 -26243.489,E2 -26243.489} C_VEL
LIN {X 0,Y 157.225,Z 637.036,A -85,B 0,C 180,E1 -26244.256,E2 -26244.256} C_VEL
LIN {X 0,Y 152.857,Z 628.091,A -85,B 0,C 180,E1 -26247.373,E2 -26247.373} C_VEL
LIN {X 0,Y 148.275,Z 619.78,A -85,B 0,C 180,E1 -26251.085,E2 -26251.085} C_VEL
LIN {X 0,Y 143.95,Z 612.902,A -85,B 0,C 180,E1 -26255.196,E2 -26255.196} C_VEL
LIN {X 0,Y 141.906,Z 609.751,A -85,B 0,C 180,E1 -26257.471,E2 -26257.471} C_VEL
LIN {X 0,Y 138.92,Z 605.377,A -85,B 0,C 180,E1 -26261.376,E2 -26261.376} C_VEL
LIN {X 0,Y 136.56,Z 602.102,A -85,B 0,C 180,E1 -26265.279,E2 -26265.279} C_VEL
LIN {X 0,Y 135.963,Z 600.91,A -85,B 0,C 180,E1 -26266.549,E2 -26266.549} C_VEL
LIN {X 0,Y 133.461,Z 597.784,A -85,B 0,C 180,E1 -26273.765,E2 -26273.765} C_VEL
LIN {X 0,Y 133.028,Z 595.543,A -85,B 0,C 180,E1 -26278.486,E2 -26278.486} C_VEL
LIN {X 0,Y 133.042,Z 595.717,A -85,B 0,C 180,E1 -26281.703,E2 -26281.703} C_VEL
LIN {X 0,Y 135.419,Z 600.526,A -85,B 0,C 180,E1 -26291.981,E2 -26291.981} C_VEL
LIN {X 0,Y 136.215,Z 601.294,A -85,B 0,C 180,E1 -26293.615,E2 -26293.615} C_VEL
LIN {X 0,Y 138.301,Z 604.736,A -85,B 0,C 180,E1 -26297.37,E2 -26297.37} C_VEL
LIN {X 0,Y 139.516,Z 606.214,A -85,B 0,C 180,E1 -26299.113,E2 -26299.113} C_VEL
LIN {X 0,Y 142.719,Z 610.993,A -85,B 0,C 180,E1 -26303.105,E2 -26303.105} C_VEL
LIN {X 0,Y 145.62,Z 615.548,A -85,B 0,C 180,E1 -26306.129,E2 -26306.129} C_VEL
LIN {X 0,Y 147.658,Z 618.987,A -85,B 0,C 180,E1 -26308.035,E2 -26308.035} C_VEL
LIN {X 0,Y 151.361,Z 627.328,A -85,B 0,C 180,E1 -26311.296,E2 -26311.296} C_VEL
LIN {X 0,Y 154.865,Z 636.269,A -85,B 0,C 180,E1 -26314.082,E2 -26314.082} C_VEL
LIN {X 0,Y 156.885,Z 642.317,A -85,B 0,C 180,E1 -26315.617,E2 -26315.617} C_VEL
LIN {X 0,Y 154.196,Z 673.05,A -85,B 0,C 180,E1 -26316.777,E2 -26316.777} C_VEL
LIN {X 0,Y 151.849,Z 686.573,A -85,B 0,C 180,E1 -26317.651,E2 -26317.651} C_VEL
LIN {X 0,Y 148.645,Z 698.526,A -85,B 0,C 180,E1 -26318.732,E2 -26318.732} C_VEL
LIN {X 0,Y 144.339,Z 711.186,A -85,B 0,C 180,E1 -26320.47,E2 -26320.47} C_VEL
LIN {X 0,Y 139.534,Z 722.441,A -85,B 0,C 180,E1 -26322.559,E2 -26322.559} C_VEL
LIN {X 0,Y 134.4,Z 732.578,A -85,B 0,C 180,E1 -26325.099,E2 -26325.099} C_VEL
LIN {X 0,Y 129.069,Z 741.721,A -85,B 0,C 180,E1 -26328.166,E2 -26328.166} C_VEL
LIN {X 0,Y 123.279,Z 750.638,A -85,B 0,C 180,E1 -26332.208,E2 -26332.208} C_VEL
LIN {X 0,Y 118.65,Z 757.216,A -85,B 0,C 180,E1 -26336.229,E2 -26336.229} C_VEL
LIN {X 0,Y 114.507,Z 762.663,A -85,B 0,C 180,E1 -26340.597,E2 -26340.597} C_VEL
LIN {X 0,Y 110.829,Z 767.377,A -85,B 0,C 180,E1 -26345.662,E2 -26345.662} C_VEL
LIN {X 0,Y 107.989,Z 770.985,A -85,B 0,C 180,E1 -26351.013,E2 -26351.013} C_VEL
LIN {X 0,Y 106.704,Z 772.848,A -85,B 0,C 180,E1 -26354.728,E2 -26354.728} C_VEL
LIN {X 0,Y 105.796,Z 774.246,A -85,B 0,C 180,E1 -26358.508,E2 -26358.508} C_VEL
LIN {X 0,Y 105.035,Z 775.857,A -85,B 0,C 180,E1 -26366.167,E2 -26366.167} C_VEL
LIN {X 0,Y 105.167,Z 776.073,A -85,B 0,C 180,E1 -26370.003,E2 -26370.003} C_VEL
LIN {X 0,Y 105.346,Z 775.848,A -85,B 0,C 180,E1 -26373.828,E2 -26373.828} C_VEL
LIN {X 0,Y 106.7,Z 774.228,A -85,B 0,C 180,E1 -26381.4,E2 -26381.4} C_VEL
LIN {X 0,Y 108.024,Z 772.825,A -85,B 0,C 180,E1 -26385.087,E2 -26385.087} C_VEL
LIN {X 0,Y 110.983,Z 769.894,A -85,B 0,C 180,E1 -26390.386,E2 -26390.386} C_VEL
LIN {X 0,Y 115.472,Z 765.977,A -85,B 0,C 180,E1 -26395.461,E2 -26395.461} C_VEL
LIN {X 0,Y 121.996,Z 772.685,A -85,B 0,C 180,E1 -26403.184,E2 -26403.184} C_VEL
LIN {X 0,Y 127.477,Z 776.029,A -85,B 0,C 180,E1 -26407.336,E2 -26407.336} C_VEL
LIN {X 0,Y 130.964,Z 777.499,A -85,B 0,C 180,E1 -26409.403,E2 -26409.403} C_VEL
LIN {X 0,Y 132.25,Z 778.07,A -85,B 0,C 180,E1 -26410.711,E2 -26410.711} C_VEL
LIN {X 0,Y 133.279,Z 778.445,A -85,B 0,C 180,E1 -26415.248,E2 -26415.248} C_VEL
LIN {X 0,Y 133.985,Z 778.602,A -85,B 0,C 180,E1 -26416.179,E2 -26416.179} C_VEL
LIN {X 0,Y 125.886,Z 775.485,A -85,B 0,C 180,E1 -26420.057,E2 -26420.057} C_VEL
LIN {X 0,Y 117.763,Z 770.429,A -85,B 0,C 180,E1 -26425.462,E2 -26425.462} C_VEL
LIN {X 0,Y 112.913,Z 765.69,A -85,B 0,C 180,E1 -26430.136,E2 -26430.136} C_VEL
LIN {X 0,Y 109.051,Z 759.616,A -85,B 0,C 180,E1 -26435.736,E2 -26435.736} C_VEL
LIN {X 0,Y 106.585,Z 751.057,A -85,B 0,C 180,E1 -26442.739,E2 -26442.739} C_VEL
LIN {X 0,Y 106.112,Z 742.495,A -85,B 0,C 180,E1 -26448.539,E2 -26448.539} C_VEL
LIN {X 0,Y 106.22,Z 735.496,A -85,B 0,C 180,E1 -26452.396,E2 -26452.396} C_VEL
LIN {X 0,Y 106.151,Z 729.036,A -85,B 0,C 180,E1 -26455.252,E2 -26455.252} C_VEL
LIN {X 0,Y 105.868,Z 717.183,A -85,B 0,C 180,E1 -26459.406,E2 -26459.406} C_VEL
LIN {X 0,Y 105.356,Z 715.844,A -85,B 0,C 180,E1 -26460.497,E2 -26460.497} C_VEL
LIN {X 0,Y 105.056,Z 715.859,A -85,B 0,C 180,E1 -26461.885,E2 -26461.885} C_VEL
LIN {X 0,Y 105.816,Z 714.886,A -85,B 0,C 180,E1 -26463.808,E2 -26463.808} C_VEL
LIN {X 0,Y 107.576,Z 712.412,A -85,B 0,C 180,E1 -26465.624,E2 -26465.624} C_VEL
LIN {X 0,Y 109.652,Z 710.26,A -85,B 0,C 180,E1 -26469.223,E2 -26469.223} C_VEL
LIN {X 0,Y 111.444,Z 708.032,A -85,B 0,C 180,E1 -26470.906,E2 -26470.906} C_VEL
LIN {X 0,Y 113.911,Z 704.683,A -85,B 0,C 180,E1 -26472.574,E2 -26472.574} C_VEL
LIN {X 0,Y 115.195,Z 703.556,A -85,B 0,C 180,E1 -26474.125,E2 -26474.125} C_VEL
LIN {X 0,Y 117.94,Z 700.245,A -85,B 0,C 180,E1 -26476.207,E2 -26476.207} C_VEL
LIN {X 0,Y 121.181,Z 695.552,A -85,B 0,C 180,E1 -26477.904,E2 -26477.904} C_VEL
LIN {X 0,Y 123.047,Z 692.293,A -85,B 0,C 180,E1 -26478.658,E2 -26478.658} C_VEL
LIN {X 0,Y 125.748,Z 689.119,A -85,B 0,C 180,E1 -26480.531,E2 -26480.531} C_VEL
LIN {X 0,Y 129.249,Z 683.772,A -85,B 0,C 180,E1 -26482.373,E2 -26482.373} C_VEL
LIN {X 0,Y 132.385,Z 677.473,A -85,B 0,C 180,E1 -26483.619,E2 -26483.619} C_VEL
LIN {X 0,Y 135.846,Z 668.367,A -85,B 0,C 180,E1 -26484.857,E2 -26484.857} C_VEL
LIN {X 0,Y 136.707,Z 665.827,A -85,B 0,C 180,E1 -26485.197,E2 -26485.197} C_VEL
LIN {X 0,Y 139.537,Z 660.977,A -85,B 0,C 180,E1 -26486.956,E2 -26486.956} C_VEL
LIN {X 0,Y 142.684,Z 653.587,A -85,B 0,C 180,E1 -26488.608,E2 -26488.608} C_VEL
LIN {X 0,Y 144.871,Z 647.33,A -85,B 0,C 180,E1 -26489.555,E2 -26489.555} C_VEL
LIN {X 0,Y 148.633,Z 643.137,A -85,B 0,C 180,E1 -26491.663,E2 -26491.663} C_VEL
LIN {X 0,Y 152.647,Z 640.795,A -85,B 0,C 180,E1 -26493.853,E2 -26493.853} C_VEL
LIN {X 0,Y 150.879,Z 661.922,A -85,B 0,C 180,E1 -26494.635,E2 -26494.635} C_VEL
LIN {X 0,Y 149.105,Z 674.613,A -85,B 0,C 180,E1 -26495.266,E2 -26495.266} C_VEL
LIN {X 0,Y 146.293,Z 687.97,A -85,B 0,C 180,E1 -26496.417,E2 -26496.417} C_VEL
LIN {X 0,Y 142.523,Z 700.268,A -85,B 0,C 180,E1 -26497.906,E2 -26497.906} C_VEL
LIN {X 0,Y 138.193,Z 711.327,A -85,B 0,C 180,E1 -26499.714,E2 -26499.714} C_VEL
LIN {X 0,Y 133.436,Z 721.455,A -85,B 0,C 180,E1 -26501.927,E2 -26501.927} C_VEL
LIN {X 0,Y 128.31,Z 730.757,A -85,B 0,C 180,E1 -26504.594,E2 -26504.594} C_VEL
LIN {X 0,Y 122.172,Z 740.469,A -85,B 0,C 180,E1 -26508.403,E2 -26508.403} C_VEL
LIN {X 0,Y 116.358,Z 748.686,A -85,B 0,C 180,E1 -26512.84,E2 -26512.84} C_VEL
LIN {X 0,Y 111.214,Z 755.091,A -85,B 0,C 180,E1 -26517.507,E2 -26517.507} C_VEL
LIN {X 0,Y 106.822,Z 760.171,A -85,B 0,C 180,E1 -26522.575,E2 -26522.575} C_VEL
LIN {X 0,Y 103.317,Z 764.107,A -85,B 0,C 180,E1 -26528.026,E2 -26528.026} C_VEL
LIN {X 0,Y 100.717,Z 767.01,A -85,B 0,C 180,E1 -26533.789,E2 -26533.789} C_VEL
LIN {X 0,Y 99.514,Z 768.396,A -85,B 0,C 180,E1 -26537.765,E2 -26537.765} C_VEL
LIN {X 0,Y 98.704,Z 769.381,A -85,B 0,C 180,E1 -26541.81,E2 -26541.81} C_VEL
LIN {X 0,Y 98.26,Z 769.986,A -85,B 0,C 180,E1 -26545.895,E2 -26545.895} C_VEL
LIN {X 0,Y 98.152,Z 770.21,A -85,B 0,C 180,E1 -26549.996,E2 -26549.996} C_VEL
LIN {X 0,Y 98.259,Z 770.015,A -85,B 0,C 180,E1 -26554.098,E2 -26554.098} C_VEL
LIN {X 0,Y 98.703,Z 769.431,A -85,B 0,C 180,E1 -26558.184,E2 -26558.184} C_VEL
LIN {X 0,Y 100.709,Z 767.109,A -85,B 0,C 180,E1 -26566.205,E2 -26566.205} C_VEL
LIN {X 0,Y 103.288,Z 764.238,A -85,B 0,C 180,E1 -26571.973,E2 -26571.973} C_VEL
LIN {X 0,Y 106.748,Z 760.341,A -85,B 0,C 180,E1 -26577.439,E2 -26577.439} C_VEL
LIN {X 0,Y 111.134,Z 755.315,A -85,B 0,C 180,E1 -26582.512,E2 -26582.512} C_VEL
LIN {X 0,Y 116.267,Z 748.98,A -85,B 0,C 180,E1 -26587.187,E2 -26587.187} C_VEL
LIN {X 0,Y 121.752,Z 741.346,A -85,B 0,C 180,E1 -26591.373,E2 -26591.373} C_VEL
LIN {X 0,Y 127.149,Z 732.98,A -85,B 0,C 180,E1 -26594.804,E2 -26594.804} C_VEL
LIN {X 0,Y 132.759,Z 723.116,A -85,B 0,C 180,E1 -26597.824,E2 -26597.824} C_VEL
LIN {X 0,Y 138.134,Z 712.001,A -85,B 0,C 180,E1 -26600.308,E2 -26600.308} C_VEL
LIN {X 0,Y 142.453,Z 701.1,A -85,B 0,C 180,E1 -26602.122,E2 -26602.122} C_VEL
LIN {X 0,Y 146.228,Z 689.036,A -85,B 0,C 180,E1 -26603.609,E2 -26603.609} C_VEL
LIN {X 0,Y 149.09,Z 676.346,A -85,B 0,C 180,E1 -26604.73,E2 -26604.73} C_VEL
LIN {X 0,Y 150.937,Z 663.649,A -85,B 0,C 180,E1 -26605.433,E2 -26605.433} C_VEL
LIN {X 0,Y 152.965,Z 640.726,A -85,B 0,C 180,E1 -26606.244,E2 -26606.244} C_VEL
LIN {X 0,Y 152.73,Z 639.475,A -85,B 0,C 180,E1 -26606.482,E2 -26606.482} C_VEL
LIN {X 0,Y 148.135,Z 630.05,A -85,B 0,C 180,E1 -26610.182,E2 -26610.182} C_VEL
LIN {X 0,Y 144.493,Z 623.375,A -85,B 0,C 180,E1 -26613.554,E2 -26613.554} C_VEL
LIN {X 0,Y 140.299,Z 616.419,A -85,B 0,C 180,E1 -26618.199,E2 -26618.199} C_VEL
LIN {X 0,Y 137.336,Z 611.977,A -85,B 0,C 180,E1 -26622.311,E2 -26622.311} C_VEL
LIN {X 0,Y 135.062,Z 608.459,A -85,B 0,C 180,E1 -26626.458,E2 -26626.458} C_VEL
LIN {X 0,Y 134.572,Z 607.671,A -85,B 0,C 180,E1 -26627.559,E2 -26627.559} C_VEL
LIN {X 0,Y 132.148,Z 602.8,A -85,B 0,C 180,E1 -26638.289,E2 -26638.289} C_VEL
LIN {X 0,Y 132.143,Z 602.558,A -85,B 0,C 180,E1 -26640.627,E2 -26640.627} C_VEL
LIN {X 0,Y 134.958,Z 608.174,A -85,B 0,C 180,E1 -26652.93,E2 -26652.93} C_VEL
LIN {X 0,Y 137.07,Z 611.68,A -85,B 0,C 180,E1 -26656.92,E2 -26656.92} C_VEL
LIN {X 0,Y 138.07,Z 613.127,A -85,B 0,C 180,E1 -26658.454,E2 -26658.454} C_VEL
LIN {X 0,Y 140.947,Z 617.595,A -85,B 0,C 180,E1 -26662.25,E2 -26662.25} C_VEL
LIN {X 0,Y 143.757,Z 622.225,A -85,B 0,C 180,E1 -26665.355,E2 -26665.355} C_VEL
LIN {X 0,Y 145.427,Z 625.411,A -85,B 0,C 180,E1 -26667.038,E2 -26667.038} C_VEL
LIN {X 0,Y 149.137,Z 634.442,A -85,B 0,C 180,E1 -26670.535,E2 -26670.535} C_VEL
LIN {X 0,Y 152.196,Z 643.23,A -85,B 0,C 180,E1 -26673.168,E2 -26673.168} C_VEL
LIN {X 0,Y 152.634,Z 644.725,A -85,B 0,C 180,E1 -26673.541,E2 -26673.541} C_VEL
LIN {X 0,Y 150.102,Z 672.533,A -85,B 0,C 180,E1 -26674.59,E2 -26674.59} C_VEL
LIN {X 0,Y 147.631,Z 686.282,A -85,B 0,C 180,E1 -26675.457,E2 -26675.457} C_VEL
LIN {X 0,Y 144.312,Z 698.328,A -85,B 0,C 180,E1 -26676.534,E2 -26676.534} C_VEL
LIN {X 0,Y 139.843,Z 710.987,A -85,B 0,C 180,E1 -26678.26,E2 -26678.26} C_VEL
LIN {X 0,Y 134.825,Z 722.24,A -85,B 0,C 180,E1 -26680.333,E2 -26680.333} C_VEL
LIN {X 0,Y 129.47,Z 732.377,A -85,B 0,C 180,E1 -26682.881,E2 -26682.881} C_VEL
LIN {X 0,Y 123.84,Z 741.518,A -85,B 0,C 180,E1 -26685.962,E2 -26685.962} C_VEL
LIN {X 0,Y 117.722,Z 750.435,A -85,B 0,C 180,E1 -26690.08,E2 -26690.08} C_VEL
LIN {X 0,Y 112.337,Z 757.597,A -85,B 0,C 180,E1 -26694.629,E2 -26694.629} C_VEL
LIN {X 0,Y 108.368,Z 762.459,A -85,B 0,C 180,E1 -26698.751,E2 -26698.751} C_VEL
LIN {X 0,Y 104.366,Z 767.173,A -85,B 0,C 180,E1 -26704.046,E2 -26704.046} C_VEL
LIN {X 0,Y 101.259,Z 770.78,A -85,B 0,C 180,E1 -26709.698,E2 -26709.698} C_VEL
LIN {X 0,Y 99.829,Z 772.643,A -85,B 0,C 180,E1 -26713.648,E2 -26713.648} C_VEL
LIN {X 0,Y 98.811,Z 774.041,A -85,B 0,C 180,E1 -26717.683,E2 -26717.683} C_VEL
LIN {X 0,Y 98.185,Z 775.041,A -85,B 0,C 180,E1 -26721.773,E2 -26721.773} C_VEL
LIN {X 0,Y 97.941,Z 775.652,A -85,B 0,C 180,E1 -26725.889,E2 -26725.889} C_VEL
LIN {X 0,Y 98.073,Z 775.869,A -85,B 0,C 180,E1 -26730.004,E2 -26730.004} C_VEL
LIN {X 0,Y 98.263,Z 775.643,A -85,B 0,C 180,E1 -26734.105,E2 -26734.105} C_VEL
LIN {X 0,Y 98.823,Z 775.028,A -85,B 0,C 180,E1 -26738.181,E2 -26738.181} C_VEL
LIN {X 0,Y 101.192,Z 772.619,A -85,B 0,C 180,E1 -26746.133,E2 -26746.133} C_VEL
LIN {X 0,Y 104.366,Z 769.689,A -85,B 0,C 180,E1 -26751.742,E2 -26751.742} C_VEL
LIN {X 0,Y 110.703,Z 764.421,A -85,B 0,C 180,E1 -26758.437,E2 -26758.437} C_VEL
LIN {X 0,Y 118.203,Z 771.574,A -85,B 0,C 180,E1 -26766.485,E2 -26766.485} C_VEL
LIN {X 0,Y 126.519,Z 776.05,A -85,B 0,C 180,E1 -26771.807,E2 -26771.807} C_VEL
LIN {X 0,Y 133.056,Z 778.393,A -85,B 0,C 180,E1 -26774.941,E2 -26774.941} C_VEL
LIN {X 0,Y 133.279,Z 778.445,A -85,B 0,C 180,E1 -26775.248,E2 -26775.248} C_VEL
LIN {X 0,Y 133.096,Z 778.37,A -85,B 0,C 180,E1 -26776.023,E2 -26776.023} C_VEL
LIN {X 0,Y 131.62,Z 777.851,A -85,B 0,C 180,E1 -26776.867,E2 -26776.867} C_VEL
LIN {X 0,Y 128.503,Z 776.693,A -85,B 0,C 180,E1 -26777.719,E2 -26777.719} C_VEL
LIN {X 0,Y 119.542,Z 772.694,A -85,B 0,C 180,E1 -26779.236,E2 -26779.236} C_VEL
LIN {X 0,Y 116.736,Z 771.041,A -85,B 0,C 180,E1 -26780.386,E2 -26780.386} C_VEL
LIN {X 0,Y 110.577,Z 766.189,A -85,B 0,C 180,E1 -26785.109,E2 -26785.109} C_VEL
LIN {X 0,Y 105.968,Z 760.756,A -85,B 0,C 180,E1 -26790.171,E2 -26790.171} C_VEL
LIN {X 0,Y 102.283,Z 753.256,A -85,B 0,C 180,E1 -26796.729,E2 -26796.729} C_VEL
LIN {X 0,Y 100.698,Z 745.52,A -85,B 0,C 180,E1 -26802.745,E2 -26802.745} C_VEL
LIN {X 0,Y 100.415,Z 736.834,A -85,B 0,C 180,E1 -26808.494,E2 -26808.494} C_VEL
LIN {X 0,Y 100.418,Z 728.899,A -85,B 0,C 180,E1 -26812.509,E2 -26812.509} C_VEL
LIN {X 0,Y 100.067,Z 725.648,A -85,B 0,C 180,E1 -26814.094,E2 -26814.094} C_VEL
LIN {X 0,Y 99.368,Z 724.701,A -85,B 0,C 180,E1 -26815.354,E2 -26815.354} C_VEL
LIN {X 0,Y 99.138,Z 724.755,A -85,B 0,C 180,E1 -26815.935,E2 -26815.935} C_VEL
LIN {X 0,Y 102.648,Z 719.961,A -85,B 0,C 180,E1 -26825.895,E2 -26825.895} C_VEL
LIN {X 0,Y 104.459,Z 717.772,A -85,B 0,C 180,E1 -26827.733,E2 -26827.733} C_VEL
LIN {X 0,Y 107.027,Z 715.453,A -85,B 0,C 180,E1 -26831.362,E2 -26831.362} C_VEL
LIN {X 0,Y 108.763,Z 713.693,A -85,B 0,C 180,E1 -26832.881,E2 -26832.881} C_VEL
LIN {X 0,Y 111.427,Z 710.635,A -85,B 0,C 180,E1 -26834.613,E2 -26834.613} C_VEL
LIN {X 0,Y 115.348,Z 706.827,A -85,B 0,C 180,E1 -26837.737,E2 -26837.737} C_VEL
LIN {X 0,Y 118.751,Z 702.88,A -85,B 0,C 180,E1 -26839.619,E2 -26839.619} C_VEL
LIN {X 0,Y 122.312,Z 697.972,A -85,B 0,C 180,E1 -26841.047,E2 -26841.047} C_VEL
LIN {X 0,Y 123.638,Z 696.253,A -85,B 0,C 180,E1 -26841.684,E2 -26841.684} C_VEL
LIN {X 0,Y 127.379,Z 691.854,A -85,B 0,C 180,E1 -26843.713,E2 -26843.713} C_VEL
LIN {X 0,Y 131.387,Z 685.88,A -85,B 0,C 180,E1 -26845.336,E2 -26845.336} C_VEL
LIN {X 0,Y 135.593,Z 677.703,A -85,B 0,C 180,E1 -26846.657,E2 -26846.657} C_VEL
LIN {X 0,Y 138.618,Z 670.071,A -85,B 0,C 180,E1 -26847.558,E2 -26847.558} C_VEL
LIN {X 0,Y 141.95,Z 664.597,A -85,B 0,C 180,E1 -26849.27,E2 -26849.27} C_VEL
LIN {X 0,Y 145.478,Z 656.743,A -85,B 0,C 180,E1 -26850.883,E2 -26850.883} C_VEL
LIN {X 0,Y 147.203,Z 652.174,A -85,B 0,C 180,E1 -26851.58,E2 -26851.58} C_VEL
LIN {X 0,Y 147.903,Z 651.422,A -85,B 0,C 180,E1 -26851.955,E2 -26851.955} C_VEL
LIN {X 0,Y 146.523,Z 665.928,A -85,B 0,C 180,E1 -26852.491,E2 -26852.491} C_VEL
LIN {X 0,Y 144.292,Z 679.235,A -85,B 0,C 180,E1 -26853.31,E2 -26853.31} C_VEL
LIN {X 0,Y 140.899,Z 692.704,A -85,B 0,C 180,E1 -26854.608,E2 -26854.608} C_VEL
LIN {X 0,Y 137.003,Z 703.963,A -85,B 0,C 180,E1 -26856.1,E2 -26856.1} C_VEL
LIN {X 0,Y 131.88,Z 715.58,A -85,B 0,C 180,E1 -26858.18,E2 -26858.18} C_VEL
LIN {X 0,Y 126.391,Z 726.016,A -85,B 0,C 180,E1 -26860.742,E2 -26860.742} C_VEL
LIN {X 0,Y 121.148,Z 734.54,A -85,B 0,C 180,E1 -26863.516,E2 -26863.516} C_VEL
LIN {X 0,Y 115.406,Z 742.88,A -85,B 0,C 180,E1 -26867.16,E2 -26867.16} C_VEL
LIN {X 0,Y 109.844,Z 750.055,A -85,B 0,C 180,E1 -26871.401,E2 -26871.401} C_VEL
LIN {X 0,Y 103.589,Z 757.105,A -85,B 0,C 180,E1 -26877.125,E2 -26877.125} C_VEL
LIN {X 0,Y 99.24,Z 761.79,A -85,B 0,C 180,E1 -26882.589,E2 -26882.589} C_VEL
LIN {X 0,Y 95.702,Z 765.369,A -85,B 0,C 180,E1 -26888.454,E2 -26888.454} C_VEL
LIN {X 0,Y 93.918,Z 767.216,A -85,B 0,C 180,E1 -26892.579,E2 -26892.579} C_VEL
LIN {X 0,Y 92.582,Z 768.601,A -85,B 0,C 180,E1 -26896.833,E2 -26896.833} C_VEL
LIN {X 0,Y 91.694,Z 769.586,A -85,B 0,C 180,E1 -26901.178,E2 -26901.178} C_VEL
LIN {X 0,Y 91.205,Z 770.19,A -85,B 0,C 180,E1 -26905.577,E2 -26905.577} C_VEL
LIN {X 0,Y 91.058,Z 770.415,A -85,B 0,C 180,E1 -26909.996,E2 -26909.996} C_VEL
LIN {X 0,Y 91.185,Z 770.219,A -85,B 0,C 180,E1 -26914.417,E2 -26914.417} C_VEL
LIN {X 0,Y 91.692,Z 769.635,A -85,B 0,C 180,E1 -26918.814,E2 -26918.814} C_VEL
LIN {X 0,Y 93.91,Z 767.313,A -85,B 0,C 180,E1 -26927.415,E2 -26927.415} C_VEL
LIN {X 0,Y 96.749,Z 764.441,A -85,B 0,C 180,E1 -26933.545,E2 -26933.545} C_VEL
LIN {X 0,Y 100.485,Z 760.545,A -85,B 0,C 180,E1 -26939.309,E2 -26939.309} C_VEL
LIN {X 0,Y 105.224,Z 755.518,A -85,B 0,C 180,E1 -26944.587,E2 -26944.587} C_VEL
LIN {X 0,Y 110.686,Z 749.183,A -85,B 0,C 180,E1 -26949.412,E2 -26949.412} C_VEL
LIN {X 0,Y 116.23,Z 741.963,A -85,B 0,C 180,E1 -26953.481,E2 -26953.481} C_VEL
LIN {X 0,Y 122.214,Z 733.182,A -85,B 0,C 180,E1 -26957.15,E2 -26957.15} C_VEL
LIN {X 0,Y 128.113,Z 723.316,A -85,B 0,C 180,E1 -26960.171,E2 -26960.171} C_VEL
LIN {X 0,Y 133.723,Z 712.201,A -85,B 0,C 180,E1 -26962.642,E2 -26962.642} C_VEL
LIN {X 0,Y 138.215,Z 701.299,A -85,B 0,C 180,E1 -26964.442,E2 -26964.442} C_VEL
LIN {X 0,Y 142.138,Z 689.233,A -85,B 0,C 180,E1 -26965.909,E2 -26965.909} C_VEL
LIN {X 0,Y 145.06,Z 676.772,A -85,B 0,C 180,E1 -26967.006,E2 -26967.006} C_VEL
LIN {X 0,Y 147.001,Z 664.076,A -85,B 0,C 180,E1 -26967.7,E2 -26967.7} C_VEL
LIN {X 0,Y 148.913,Z 643.134,A -85,B 0,C 180,E1 -26968.451,E2 -26968.451} C_VEL
LIN {X 0,Y 144.877,Z 634.471,A -85,B 0,C 180,E1 -26972.068,E2 -26972.068} C_VEL
LIN {X 0,Y 141.488,Z 628.157,A -85,B 0,C 180,E1 -26975.553,E2 -26975.553} C_VEL
LIN {X 0,Y 138.244,Z 622.544,A -85,B 0,C 180,E1 -26979.542,E2 -26979.542} C_VEL
LIN {X 0,Y 135.791,Z 618.57,A -85,B 0,C 180,E1 -26983.268,E2 -26983.268} C_VEL
LIN {X 0,Y 133.428,Z 614.538,A -85,B 0,C 180,E1 -26988.126,E2 -26988.126} C_VEL
LIN {X 0,Y 131.275,Z 609.574,A -85,B 0,C 180,E1 -26999.282,E2 -26999.282} C_VEL
LIN {X 0,Y 131.261,Z 609.974,A -85,B 0,C 180,E1 -27001.262,E2 -27001.262} C_VEL
LIN {X 0,Y 133.684,Z 614.97,A -85,B 0,C 180,E1 -27012.139,E2 -27012.139} C_VEL
LIN {X 0,Y 136.369,Z 619.503,A -85,B 0,C 180,E1 -27017.331,E2 -27017.331} C_VEL
LIN {X 0,Y 139.005,Z 623.863,A -85,B 0,C 180,E1 -27021.115,E2 -27021.115} C_VEL
LIN {X 0,Y 142.18,Z 629.345,A -85,B 0,C 180,E1 -27024.837,E2 -27024.837} C_VEL
LIN {X 0,Y 145.19,Z 636.974,A -85,B 0,C 180,E1 -27028.063,E2 -27028.063} C_VEL
LIN {X 0,Y 148.175,Z 645.696,A -85,B 0,C 180,E1 -27030.952,E2 -27030.952} C_VEL
LIN {X 0,Y 148.597,Z 647.116,A -85,B 0,C 180,E1 -27031.349,E2 -27031.349} C_VEL
LIN {X 0,Y 146.104,Z 672.958,A -85,B 0,C 180,E1 -27032.333,E2 -27032.333} C_VEL
LIN {X 0,Y 143.531,Z 686.533,A -85,B 0,C 180,E1 -27033.184,E2 -27033.184} C_VEL
LIN {X 0,Y 140.206,Z 698.13,A -85,B 0,C 180,E1 -27034.205,E2 -27034.205} C_VEL
LIN {X 0,Y 135.566,Z 710.787,A -85,B 0,C 180,E1 -27035.906,E2 -27035.906} C_VEL
LIN {X 0,Y 130.343,Z 722.039,A -85,B 0,C 180,E1 -27037.953,E2 -27037.953} C_VEL
LIN {X 0,Y 124.751,Z 732.175,A -85,B 0,C 180,E1 -27040.493,E2 -27040.493} C_VEL
LIN {X 0,Y 118.819,Z 741.315,A -85,B 0,C 180,E1 -27043.572,E2 -27043.572} C_VEL
LIN {X 0,Y 112.346,Z 750.231,A -85,B 0,C 180,E1 -27047.745,E2 -27047.745} C_VEL
LIN {X 0,Y 107.176,Z 756.692,A -85,B 0,C 180,E1 -27051.896,E2 -27051.896} C_VEL
LIN {X 0,Y 102.358,Z 762.256,A -85,B 0,C 180,E1 -27056.686,E2 -27056.686} C_VEL
LIN {X 0,Y 98.005,Z 766.968,A -85,B 0,C 180,E1 -27062.221,E2 -27062.221} C_VEL
LIN {X 0,Y 94.595,Z 770.575,A -85,B 0,C 180,E1 -27068.197,E2 -27068.197} C_VEL
LIN {X 0,Y 93.003,Z 772.438,A -85,B 0,C 180,E1 -27072.41,E2 -27072.41} C_VEL
LIN {X 0,Y 91.861,Z 773.836,A -85,B 0,C 180,E1 -27076.735,E2 -27076.735} C_VEL
LIN {X 0,Y 90.871,Z 775.448,A -85,B 0,C 180,E1 -27085.568,E2 -27085.568} C_VEL
LIN {X 0,Y 90.972,Z 775.664,A -85,B 0,C 180,E1 -27090.004,E2 -27090.004} C_VEL
LIN {X 0,Y 91.21,Z 775.439,A -85,B 0,C 180,E1 -27094.423,E2 -27094.423} C_VEL
LIN {X 0,Y 91.813,Z 774.823,A -85,B 0,C 180,E1 -27098.81,E2 -27098.81} C_VEL
LIN {X 0,Y 94.391,Z 772.414,A -85,B 0,C 180,E1 -27107.331,E2 -27107.331} C_VEL
LIN {X 0,Y 97.822,Z 769.484,A -85,B 0,C 180,E1 -27113.279,E2 -27113.279} C_VEL
LIN {X 0,Y 102.615,Z 765.531,A -85,B 0,C 180,E1 -27118.651,E2 -27118.651} C_VEL
LIN {X 0,Y 106.266,Z 762.761,A -85,B 0,C 180,E1 -27121.669,E2 -27121.669} C_VEL
LIN {X 0,Y 107.212,Z 763.538,A -85,B 0,C 180,E1 -27122.742,E2 -27122.742} C_VEL
LIN {X 0,Y 113.004,Z 768.885,A -85,B 0,C 180,E1 -27128.461,E2 -27128.461} C_VEL
LIN {X 0,Y 119.257,Z 772.824,A -85,B 0,C 180,E1 -27132.668,E2 -27132.668} C_VEL
LIN {X 0,Y 123.349,Z 774.762,A -85,B 0,C 180,E1 -27134.851,E2 -27134.851} C_VEL
LIN {X 0,Y 124.136,Z 775.081,A -85,B 0,C 180,E1 -27136.218,E2 -27136.218} C_VEL
LIN {X 0,Y 116.736,Z 771.041,A -85,B 0,C 180,E1 -27140.386,E2 -27140.386} C_VEL
LIN {X 0,Y 113.16,Z 768.613,A -85,B 0,C 180,E1 -27142.37,E2 -27142.37} C_VEL
LIN {X 0,Y 106.783,Z 763.503,A -85,B 0,C 180,E1 -27145.276,E2 -27145.276} C_VEL
LIN {X 0,Y 101.177,Z 757.792,A -85,B 0,C 180,E1 -27148.497,E2 -27148.497} C_VEL
LIN {X 0,Y 98.938,Z 754.338,A -85,B 0,C 180,E1 -27150.978,E2 -27150.978} C_VEL
LIN {X 0,Y 95.848,Z 745.385,A -85,B 0,C 180,E1 -27158.493,E2 -27158.493} C_VEL
LIN {X 0,Y 94.851,Z 735.2,A -85,B 0,C 180,E1 -27165.794,E2 -27165.794} C_VEL
LIN {X 0,Y 94.19,Z 733.566,A -85,B 0,C 180,E1 -27167.571,E2 -27167.571} C_VEL
LIN {X 0,Y 93.526,Z 733.351,A -85,B 0,C 180,E1 -27169.17,E2 -27169.17} C_VEL
LIN {X 0,Y 93.41,Z 732.741,A -85,B 0,C 180,E1 -27171.346,E2 -27171.346} C_VEL
LIN {X 0,Y 94.665,Z 730.233,A -85,B 0,C 180,E1 -27175.743,E2 -27175.743} C_VEL
LIN {X 0,Y 97.078,Z 726.936,A -85,B 0,C 180,E1 -27184.152,E2 -27184.152} C_VEL
LIN {X 0,Y 99.407,Z 724.81,A -85,B 0,C 180,E1 -27188.176,E2 -27188.176} C_VEL
LIN {X 0,Y 101.135,Z 723.057,A -85,B 0,C 180,E1 -27189.803,E2 -27189.803} C_VEL
LIN {X 0,Y 104.356,Z 720.493,A -85,B 0,C 180,E1 -27193.633,E2 -27193.633} C_VEL
LIN {X 0,Y 107.666,Z 717.41,A -85,B 0,C 180,E1 -27196.108,E2 -27196.108} C_VEL
LIN {X 0,Y 110.966,Z 714.337,A -85,B 0,C 180,E1 -27198.183,E2 -27198.183} C_VEL
LIN {X 0,Y 113.479,Z 712.159,A -85,B 0,C 180,E1 -27199.915,E2 -27199.915} C_VEL
LIN {X 0,Y 118.006,Z 707.595,A -85,B 0,C 180,E1 -27202.174,E2 -27202.174} C_VEL
LIN {X 0,Y 123.102,Z 701.37,A -85,B 0,C 180,E1 -27204.007,E2 -27204.007} C_VEL
LIN {X 0,Y 127.691,Z 696.479,A -85,B 0,C 180,E1 -27206.124,E2 -27206.124} C_VEL
LIN {X 0,Y 132.373,Z 690.235,A -85,B 0,C 180,E1 -27207.757,E2 -27207.757} C_VEL
LIN {X 0,Y 136.996,Z 682.285,A -85,B 0,C 180,E1 -27208.999,E2 -27208.999} C_VEL
LIN {X 0,Y 140.805,Z 673.97,A -85,B 0,C 180,E1 -27209.943,E2 -27209.943} C_VEL
LIN {X 0,Y 141.852,Z 672.52,A -85,B 0,C 180,E1 -27210.401,E2 -27210.401} C_VEL
LIN {X 0,Y 139.1,Z 685.543,A -85,B 0,C 180,E1 -27211.424,E2 -27211.424} C_VEL
LIN {X 0,Y 135.569,Z 697.169,A -85,B 0,C 180,E1 -27212.672,E2 -27212.672} C_VEL
LIN {X 0,Y 130.94,Z 708.89,A -85,B 0,C 180,E1 -27214.384,E2 -27214.384} C_VEL
LIN {X 0,Y 125.717,Z 719.529,A -85,B 0,C 180,E1 -27216.52,E2 -27216.52} C_VEL
LIN {X 0,Y 120.001,Z 729.23,A -85,B 0,C 180,E1 -27219.1,E2 -27219.1} C_VEL
LIN {X 0,Y 113.285,Z 739.099,A -85,B 0,C 180,E1 -27222.738,E2 -27222.738} C_VEL
LIN {X 0,Y 106.435,Z 747.874,A -85,B 0,C 180,E1 -27227.401,E2 -27227.401} C_VEL
LIN {X 0,Y 101.421,Z 753.506,A -85,B 0,C 180,E1 -27231.412,E2 -27231.412} C_VEL
LIN {X 0,Y 96.028,Z 758.999,A -85,B 0,C 180,E1 -27236.704,E2 -27236.704} C_VEL
LIN {X 0,Y 91.608,Z 763.301,A -85,B 0,C 180,E1 -27242.589,E2 -27242.589} C_VEL
LIN {X 0,Y 89.143,Z 765.575,A -85,B 0,C 180,E1 -27246.78,E2 -27246.78} C_VEL
LIN {X 0,Y 87.177,Z 767.421,A -85,B 0,C 180,E1 -27251.184,E2 -27251.184} C_VEL
LIN {X 0,Y 84.681,Z 769.791,A -85,B 0,C 180,E1 -27260.441,E2 -27260.441} C_VEL
LIN {X 0,Y 84.125,Z 770.395,A -85,B 0,C 180,E1 -27265.204,E2 -27265.204} C_VEL
LIN {X 0,Y 83.975,Z 770.619,A -85,B 0,C 180,E1 -27269.996,E2 -27269.996} C_VEL
LIN {X 0,Y 84.107,Z 770.424,A -85,B 0,C 180,E1 -27274.789,E2 -27274.789} C_VEL
LIN {X 0,Y 84.678,Z 769.839,A -85,B 0,C 180,E1 -27279.551,E2 -27279.551} C_VEL
LIN {X 0,Y 87.168,Z 767.517,A -85,B 0,C 180,E1 -27288.81,E2 -27288.81} C_VEL
LIN {X 0,Y 90.278,Z 764.645,A -85,B 0,C 180,E1 -27295.347,E2 -27295.347} C_VEL
LIN {X 0,Y 94.345,Z 760.749,A -85,B 0,C 180,E1 -27301.425,E2 -27301.425} C_VEL
LIN {X 0,Y 99.459,Z 755.721,A -85,B 0,C 180,E1 -27306.91,E2 -27306.91} C_VEL
LIN {X 0,Y 105.287,Z 749.386,A -85,B 0,C 180,E1 -27311.87,E2 -27311.87} C_VEL
LIN {X 0,Y 111.494,Z 741.758,A -85,B 0,C 180,E1 -27316.194,E2 -27316.194} C_VEL
LIN {X 0,Y 117.508,Z 733.383,A -85,B 0,C 180,E1 -27319.686,E2 -27319.686} C_VEL
LIN {X 0,Y 123.702,Z 723.517,A -85,B 0,C 180,E1 -27322.688,E2 -27322.688} C_VEL
LIN {X 0,Y 129.537,Z 712.401,A -85,B 0,C 180,E1 -27325.14,E2 -27325.14} C_VEL
LIN {X 0,Y 134.214,Z 701.498,A -85,B 0,C 180,E1 -27326.906,E2 -27326.906} C_VEL
LIN {X 0,Y 138.293,Z 689.43,A -85,B 0,C 180,E1 -27328.34,E2 -27328.34} C_VEL
LIN {X 0,Y 141.379,Z 676.711,A -85,B 0,C 180,E1 -27329.429,E2 -27329.429} C_VEL
LIN {X 0,Y 143.362,Z 664.104,A -85,B 0,C 180,E1 -27330.099,E2 -27330.099} C_VEL
LIN {X 0,Y 145.036,Z 646.273,A -85,B 0,C 180,E1 -27330.748,E2 -27330.748} C_VEL
LIN {X 0,Y 141.724,Z 638.893,A -85,B 0,C 180,E1 -27334.087,E2 -27334.087} C_VEL
LIN {X 0,Y 138.595,Z 632.75,A -85,B 0,C 180,E1 -27337.731,E2 -27337.731} C_VEL
LIN {X 0,Y 136.108,Z 628.353,A -85,B 0,C 180,E1 -27341.172,E2 -27341.172} C_VEL
LIN {X 0,Y 134.229,Z 625.059,A -85,B 0,C 180,E1 -27344.352,E2 -27344.352} C_VEL
LIN {X 0,Y 132.22,Z 621.361,A -85,B 0,C 180,E1 -27348.89,E2 -27348.89} C_VEL
LIN {X 0,Y 130.404,Z 616.623,A -85,B 0,C 180,E1 -27360,E2 -27360} C_VEL
LIN {X 0,Y 132.422,Z 621.708,A -85,B 0,C 180,E1 -27371.286,E2 -27371.286} C_VEL
LIN {X 0,Y 134.927,Z 626.284,A -85,B 0,C 180,E1 -27376.548,E2 -27376.548} C_VEL
LIN {X 0,Y 137.247,Z 630.342,A -85,B 0,C 180,E1 -27380.124,E2 -27380.124} C_VEL
LIN {X 0,Y 139.826,Z 635.091,A -85,B 0,C 180,E1 -27383.415,E2 -27383.415} C_VEL
LIN {X 0,Y 142.55,Z 642.557,A -85,B 0,C 180,E1 -27386.637,E2 -27386.637} C_VEL
LIN {X 0,Y 144.778,Z 649.604,A -85,B 0,C 180,E1 -27389.041,E2 -27389.041} C_VEL
LIN {X 0,Y 142.423,Z 672.876,A -85,B 0,C 180,E1 -27389.928,E2 -27389.928} C_VEL
LIN {X 0,Y 139.763,Z 686.376,A -85,B 0,C 180,E1 -27390.75,E2 -27390.75} C_VEL
LIN {X 0,Y 136.347,Z 697.932,A -85,B 0,C 180,E1 -27391.74,E2 -27391.74} C_VEL
LIN {X 0,Y 132.204,Z 709.003,A -85,B 0,C 180,E1 -27393.152,E2 -27393.152} C_VEL
LIN {X 0,Y 126.756,Z 720.544,A -85,B 0,C 180,E1 -27395.138,E2 -27395.138} C_VEL
LIN {X 0,Y 120.897,Z 730.943,A -85,B 0,C 180,E1 -27397.628,E2 -27397.628} C_VEL
LIN {X 0,Y 115.262,Z 739.448,A -85,B 0,C 180,E1 -27400.348,E2 -27400.348} C_VEL
LIN {X 0,Y 108.269,Z 748.668,A -85,B 0,C 180,E1 -27404.441,E2 -27404.441} C_VEL
LIN {X 0,Y 102.082,Z 756.036,A -85,B 0,C 180,E1 -27409.094,E2 -27409.094} C_VEL
LIN {X 0,Y 96.499,Z 762.052,A -85,B 0,C 180,E1 -27414.368,E2 -27414.368} C_VEL
LIN {X 0,Y 91.756,Z 766.764,A -85,B 0,C 180,E1 -27420.146,E2 -27420.146} C_VEL
LIN {X 0,Y 88.006,Z 770.37,A -85,B 0,C 180,E1 -27426.471,E2 -27426.471} C_VEL
LIN {X 0,Y 86.236,Z 772.233,A -85,B 0,C 180,E1 -27430.979,E2 -27430.979} C_VEL
LIN {X 0,Y 84.95,Z 773.631,A -85,B 0,C 180,E1 -27435.634,E2 -27435.634} C_VEL
LIN {X 0,Y 84.132,Z 774.632,A -85,B 0,C 180,E1 -27440.387,E2 -27440.387} C_VEL
LIN {X 0,Y 83.787,Z 775.243,A -85,B 0,C 180,E1 -27445.193,E2 -27445.193} C_VEL
LIN {X 0,Y 83.879,Z 775.459,A -85,B 0,C 180,E1 -27450.004,E2 -27450.004} C_VEL
LIN {X 0,Y 84.133,Z 775.234,A -85,B 0,C 180,E1 -27454.796,E2 -27454.796} C_VEL
LIN {X 0,Y 84.805,Z 774.618,A -85,B 0,C 180,E1 -27459.545,E2 -27459.545} C_VEL
LIN {X 0,Y 87.649,Z 772.209,A -85,B 0,C 180,E1 -27468.711,E2 -27468.711} C_VEL
LIN {X 0,Y 91.366,Z 769.279,A -85,B 0,C 180,E1 -27475.032,E2 -27475.032} C_VEL
LIN {X 0,Y 96.461,Z 765.326,A -85,B 0,C 180,E1 -27480.668,E2 -27480.668} C_VEL
LIN {X 0,Y 102.235,Z 760.984,A -85,B 0,C 180,E1 -27485.154,E2 -27485.154} C_VEL
LIN {X 0,Y 103.168,Z 761.494,A -85,B 0,C 180,E1 -27485.987,E2 -27485.987} C_VEL
LIN {X 0,Y 110.043,Z 767.525,A -85,B 0,C 180,E1 -27492.117,E2 -27492.117} C_VEL
LIN {X 0,Y 115.032,Z 770.539,A -85,B 0,C 180,E1 -27495.23,E2 -27495.23} C_VEL
LIN {X 0,Y 114.798,Z 770.352,A -85,B 0,C 180,E1 -27496.366,E2 -27496.366} C_VEL
LIN {X 0,Y 107.239,Z 764.848,A -85,B 0,C 180,E1 -27501.495,E2 -27501.495} C_VEL
LIN {X 0,Y 100.584,Z 757.339,A -85,B 0,C 180,E1 -27508.396,E2 -27508.396} C_VEL
LIN {X 0,Y 98.938,Z 754.338,A -85,B 0,C 180,E1 -27510.978,E2 -27510.978} C_VEL
LIN {X 0,Y 97.408,Z 751.863,A -85,B 0,C 180,E1 -27512.644,E2 -27512.644} C_VEL
LIN {X 0,Y 92.199,Z 745.665,A -85,B 0,C 180,E1 -27515.771,E2 -27515.771} C_VEL
LIN {X 0,Y 89.8,Z 743.266,A -85,B 0,C 180,E1 -27517.773,E2 -27517.773} C_VEL
LIN {X 0,Y 88.715,Z 742.274,A -85,B 0,C 180,E1 -27519.636,E2 -27519.636} C_VEL
LIN {X 0,Y 88.2,Z 741.808,A -85,B 0,C 180,E1 -27521.414,E2 -27521.414} C_VEL
LIN {X 0,Y 88.761,Z 739.138,A -85,B 0,C 180,E1 -27526.259,E2 -27526.259} C_VEL
LIN {X 0,Y 88.399,Z 737.949,A -85,B 0,C 180,E1 -27530.851,E2 -27530.851} C_VEL
LIN {X 0,Y 88.65,Z 737.134,A -85,B 0,C 180,E1 -27533.171,E2 -27533.171} C_VEL
LIN {X 0,Y 89.39,Z 735.919,A -85,B 0,C 180,E1 -27535.491,E2 -27535.491} C_VEL
LIN {X 0,Y 94.5,Z 730.676,A -85,B 0,C 180,E1 -27548.554,E2 -27548.554} C_VEL
LIN {X 0,Y 96.674,Z 728.975,A -85,B 0,C 180,E1 -27551.134,E2 -27551.134} C_VEL
LIN {X 0,Y 98.121,Z 727.734,A -85,B 0,C 180,E1 -27552.409,E2 -27552.409} C_VEL
LIN {X 0,Y 101.589,Z 725.347,A -85,B 0,C 180,E1 -27556.065,E2 -27556.065} C_VEL
LIN {X 0,Y 105.174,Z 722.479,A -85,B 0,C 180,E1 -27558.506,E2 -27558.506} C_VEL
LIN {X 0,Y 109.143,Z 719.187,A -85,B 0,C 180,E1 -27560.742,E2 -27560.742} C_VEL
LIN {X 0,Y 114.284,Z 715.021,A -85,B 0,C 180,E1 -27563.563,E2 -27563.563} C_VEL
LIN {X 0,Y 119.278,Z 710.199,A -85,B 0,C 180,E1 -27565.488,E2 -27565.488} C_VEL
LIN {X 0,Y 123.984,Z 705.036,A -85,B 0,C 180,E1 -27566.967,E2 -27566.967} C_VEL
LIN {X 0,Y 128.933,Z 700.05,A -85,B 0,C 180,E1 -27568.845,E2 -27568.845} C_VEL
LIN {X 0,Y 131.629,Z 696.87,A -85,B 0,C 180,E1 -27569.683,E2 -27569.683} C_VEL
LIN {X 0,Y 131.359,Z 698.822,A -85,B 0,C 180,E1 -27570.247,E2 -27570.247} C_VEL
LIN {X 0,Y 126.372,Z 710.531,A -85,B 0,C 180,E1 -27571.99,E2 -27571.99} C_VEL
LIN {X 0,Y 120.277,Z 722.08,A -85,B 0,C 180,E1 -27574.372,E2 -27574.372} C_VEL
LIN {X 0,Y 114.367,Z 731.381,A -85,B 0,C 180,E1 -27576.973,E2 -27576.973} C_VEL
LIN {X 0,Y 108.166,Z 739.85,A -85,B 0,C 180,E1 -27580.228,E2 -27580.228} C_VEL
LIN {X 0,Y 101.308,Z 748.081,A -85,B 0,C 180,E1 -27584.674,E2 -27584.674} C_VEL
LIN {X 0,Y 95.98,Z 753.712,A -85,B 0,C 180,E1 -27588.771,E2 -27588.771} C_VEL
LIN {X 0,Y 90.164,Z 759.206,A -85,B 0,C 180,E1 -27594.221,E2 -27594.221} C_VEL
LIN {X 0,Y 85.358,Z 763.507,A -85,B 0,C 180,E1 -27600.391,E2 -27600.391} C_VEL
LIN {X 0,Y 82.676,Z 765.78,A -85,B 0,C 180,E1 -27604.843,E2 -27604.843} C_VEL
LIN {X 0,Y 80.474,Z 767.627,A -85,B 0,C 180,E1 -27609.549,E2 -27609.549} C_VEL
LIN {X 0,Y 77.7,Z 769.996,A -85,B 0,C 180,E1 -27619.573,E2 -27619.573} C_VEL
LIN {X 0,Y 77.068,Z 770.599,A -85,B 0,C 180,E1 -27624.763,E2 -27624.763} C_VEL
LIN {X 0,Y 76.896,Z 770.823,A -85,B 0,C 180,E1 -27629.996,E2 -27629.996} C_VEL
LIN {X 0,Y 77.055,Z 770.628,A -85,B 0,C 180,E1 -27635.229,E2 -27635.229} C_VEL
LIN {X 0,Y 77.698,Z 770.044,A -85,B 0,C 180,E1 -27640.418,E2 -27640.418} C_VEL
LIN {X 0,Y 80.463,Z 767.722,A -85,B 0,C 180,E1 -27650.444,E2 -27650.444} C_VEL
LIN {X 0,Y 83.914,Z 764.849,A -85,B 0,C 180,E1 -27657.423,E2 -27657.423} C_VEL
LIN {X 0,Y 88.351,Z 760.953,A -85,B 0,C 180,E1 -27663.831,E2 -27663.831} C_VEL
LIN {X 0,Y 93.869,Z 755.925,A -85,B 0,C 180,E1 -27669.518,E2 -27669.518} C_VEL
LIN {X 0,Y 100.102,Z 749.59,A -85,B 0,C 180,E1 -27674.589,E2 -27674.589} C_VEL
LIN {X 0,Y 106.694,Z 741.961,A -85,B 0,C 180,E1 -27678.952,E2 -27678.952} C_VEL
LIN {X 0,Y 113.042,Z 733.585,A -85,B 0,C 180,E1 -27682.432,E2 -27682.432} C_VEL
LIN {X 0,Y 119.545,Z 723.718,A -85,B 0,C 180,E1 -27685.386,E2 -27685.386} C_VEL
LIN {X 0,Y 125.623,Z 712.601,A -85,B 0,C 180,E1 -27687.792,E2 -27687.792} C_VEL
LIN {X 0,Y 130.482,Z 701.696,A -85,B 0,C 180,E1 -27689.512,E2 -27689.512} C_VEL
LIN {X 0,Y 134.706,Z 689.627,A -85,B 0,C 180,E1 -27690.908,E2 -27690.908} C_VEL
LIN {X 0,Y 137.809,Z 677.422,A -85,B 0,C 180,E1 -27691.932,E2 -27691.932} C_VEL
LIN {X 0,Y 139.835,Z 665.405,A -85,B 0,C 180,E1 -27692.571,E2 -27692.571} C_VEL
LIN {X 0,Y 141.432,Z 649.489,A -85,B 0,C 180,E1 -27693.135,E2 -27693.135} C_VEL
LIN {X 0,Y 138.404,Z 642.584,A -85,B 0,C 180,E1 -27696.624,E2 -27696.624} C_VEL
LIN {X 0,Y 135.553,Z 636.837,A -85,B 0,C 180,E1 -27700.502,E2 -27700.502} C_VEL
LIN {X 0,Y 132.824,Z 631.703,A -85,B 0,C 180,E1 -27705.248,E2 -27705.248} C_VEL
LIN {X 0,Y 131.07,Z 628.218,A -85,B 0,C 180,E1 -27709.574,E2 -27709.574} C_VEL
LIN {X 0,Y 129.528,Z 623.759,A -85,B 0,C 180,E1 -27720,E2 -27720} C_VEL
LIN {X 0,Y 131.25,Z 628.615,A -85,B 0,C 180,E1 -27730.607,E2 -27730.607} C_VEL
LIN {X 0,Y 133.473,Z 632.959,A -85,B 0,C 180,E1 -27735.671,E2 -27735.671} C_VEL
LIN {X 0,Y 135.684,Z 637.07,A -85,B 0,C 180,E1 -27739.33,E2 -27739.33} C_VEL
LIN {X 0,Y 137.874,Z 641.689,A -85,B 0,C 180,E1 -27742.378,E2 -27742.378} C_VEL
LIN {X 0,Y 140.32,Z 649.186,A -85,B 0,C 180,E1 -27745.552,E2 -27745.552} C_VEL
LIN {X 0,Y 141.188,Z 652.266,A -85,B 0,C 180,E1 -27746.615,E2 -27746.615} C_VEL
LIN {X 0,Y 138.929,Z 673.202,A -85,B 0,C 180,E1 -27747.411,E2 -27747.411} C_VEL
LIN {X 0,Y 136.269,Z 686.166,A -85,B 0,C 180,E1 -27748.18,E2 -27748.18} C_VEL
LIN {X 0,Y 132.755,Z 697.734,A -85,B 0,C 180,E1 -27749.138,E2 -27749.138} C_VEL
LIN {X 0,Y 127.753,Z 710.388,A -85,B 0,C 180,E1 -27750.738,E2 -27750.738} C_VEL
LIN {X 0,Y 122.107,Z 721.637,A -85,B 0,C 180,E1 -27752.68,E2 -27752.68} C_VEL
LIN {X 0,Y 116.024,Z 731.771,A -85,B 0,C 180,E1 -27755.146,E2 -27755.146} C_VEL
LIN {X 0,Y 109.511,Z 740.911,A -85,B 0,C 180,E1 -27758.178,E2 -27758.178} C_VEL
LIN {X 0,Y 102.238,Z 749.824,A -85,B 0,C 180,E1 -27762.362,E2 -27762.362} C_VEL
LIN {X 0,Y 95.371,Z 757.316,A -85,B 0,C 180,E1 -27767.469,E2 -27767.469} C_VEL
LIN {X 0,Y 90.813,Z 761.849,A -85,B 0,C 180,E1 -27771.753,E2 -27771.753} C_VEL
LIN {X 0,Y 85.645,Z 766.559,A -85,B 0,C 180,E1 -27777.771,E2 -27777.771} C_VEL
LIN {X 0,Y 81.512,Z 770.165,A -85,B 0,C 180,E1 -27784.467,E2 -27784.467} C_VEL
LIN {X 0,Y 79.519,Z 772.028,A -85,B 0,C 180,E1 -27789.302,E2 -27789.302} C_VEL
LIN {X 0,Y 78.055,Z 773.426,A -85,B 0,C 180,E1 -27794.333,E2 -27794.333} C_VEL
LIN {X 0,Y 77.119,Z 774.427,A -85,B 0,C 180,E1 -27799.503,E2 -27799.503} C_VEL
LIN {X 0,Y 76.707,Z 775.039,A -85,B 0,C 180,E1 -27804.748,E2 -27804.748} C_VEL
LIN {X 0,Y 76.777,Z 775.255,A -85,B 0,C 180,E1 -27810.004,E2 -27810.004} C_VEL
LIN {X 0,Y 77.076,Z 775.03,A -85,B 0,C 180,E1 -27815.236,E2 -27815.236} C_VEL
LIN {X 0,Y 77.831,Z 774.413,A -85,B 0,C 180,E1 -27820.409,E2 -27820.409} C_VEL
LIN {X 0,Y 80.974,Z 772.004,A -85,B 0,C 180,E1 -27830.319,E2 -27830.319} C_VEL
LIN {X 0,Y 84.991,Z 769.073,A -85,B 0,C 180,E1 -27837.056,E2 -27837.056} C_VEL
LIN {X 0,Y 90.45,Z 765.121,A -85,B 0,C 180,E1 -27842.954,E2 -27842.954} C_VEL
LIN {X 0,Y 98.713,Z 759.037,A -85,B 0,C 180,E1 -27848.864,E2 -27848.864} C_VEL
LIN {X 0,Y 99.525,Z 759.256,A -85,B 0,C 180,E1 -27849.464,E2 -27849.464} C_VEL
LIN {X 0,Y 105.39,Z 764.272,A -85,B 0,C 180,E1 -27854.408,E2 -27854.408} C_VEL
LIN {X 0,Y 106.863,Z 765.303,A -85,B 0,C 180,E1 -27855.393,E2 -27855.393} C_VEL
LIN {X 0,Y 105.959,Z 764.598,A -85,B 0,C 180,E1 -27856.614,E2 -27856.614} C_VEL
LIN {X 0,Y 98.627,Z 757.73,A -85,B 0,C 180,E1 -27862.72,E2 -27862.72} C_VEL
LIN {X 0,Y 93.029,Z 748.762,A -85,B 0,C 180,E1 -27870.59,E2 -27870.59} C_VEL
LIN {X 0,Y 91.295,Z 744.48,A -85,B 0,C 180,E1 -27874.341,E2 -27874.341} C_VEL
LIN {X 0,Y 89.976,Z 742.994,A -85,B 0,C 180,E1 -27876.555,E2 -27876.555} C_VEL
LIN {X 0,Y 88.715,Z 742.274,A -85,B 0,C 180,E1 -27879.636,E2 -27879.636} C_VEL
LIN {X 0,Y 87.004,Z 741.401,A -85,B 0,C 180,E1 -27884.63,E2 -27884.63} C_VEL
LIN {X 0,Y 84.677,Z 740.486,A -85,B 0,C 180,E1 -27895.066,E2 -27895.066} C_VEL
LIN {X 0,Y 85.366,Z 739.328,A -85,B 0,C 180,E1 -27900.283,E2 -27900.283} C_VEL
LIN {X 0,Y 90.856,Z 735.161,A -85,B 0,C 180,E1 -27911.15,E2 -27911.15} C_VEL
LIN {X 0,Y 96.818,Z 731.155,A -85,B 0,C 180,E1 -27916.88,E2 -27916.88} C_VEL
LIN {X 0,Y 99.208,Z 729.724,A -85,B 0,C 180,E1 -27918.957,E2 -27918.957} C_VEL
LIN {X 0,Y 104.109,Z 726.199,A -85,B 0,C 180,E1 -27921.795,E2 -27921.795} C_VEL
LIN {X 0,Y 112.479,Z 720.125,A -85,B 0,C 180,E1 -27925.937,E2 -27925.937} C_VEL
LIN {X 0,Y 118.994,Z 714.553,A -85,B 0,C 180,E1 -27928.197,E2 -27928.197} C_VEL
LIN {X 0,Y 121.435,Z 712.081,A -85,B 0,C 180,E1 -27928.835,E2 -27928.835} C_VEL
LIN {X 0,Y 121.324,Z 713.585,A -85,B 0,C 180,E1 -27929.663,E2 -27929.663} C_VEL
LIN {X 0,Y 115.014,Z 724.508,A -85,B 0,C 180,E1 -27932.018,E2 -27932.018} C_VEL
LIN {X 0,Y 108.918,Z 733.388,A -85,B 0,C 180,E1 -27934.639,E2 -27934.639} C_VEL
LIN {X 0,Y 102.207,Z 741.831,A -85,B 0,C 180,E1 -27938.059,E2 -27938.059} C_VEL
LIN {X 0,Y 95.258,Z 749.513,A -85,B 0,C 180,E1 -27942.452,E2 -27942.452} C_VEL
LIN {X 0,Y 88.61,Z 755.915,A -85,B 0,C 180,E1 -27947.606,E2 -27947.606} C_VEL
LIN {X 0,Y 82.604,Z 760.996,A -85,B 0,C 180,E1 -27953.443,E2 -27953.443} C_VEL
LIN {X 0,Y 77.701,Z 764.93,A -85,B 0,C 180,E1 -27960.162,E2 -27960.162} C_VEL
LIN {X 0,Y 73.858,Z 767.832,A -85,B 0,C 180,E1 -27967.623,E2 -27967.623} C_VEL
LIN {X 0,Y 72.008,Z 769.216,A -85,B 0,C 180,E1 -27972.969,E2 -27972.969} C_VEL
LIN {X 0,Y 70.008,Z 770.804,A -85,B 0,C 180,E1 -27984.234,E2 -27984.234} C_VEL
LIN {X 0,Y 69.815,Z 771.027,A -85,B 0,C 180,E1 -27989.995,E2 -27989.995} C_VEL
LIN {X 0,Y 69.999,Z 770.832,A -85,B 0,C 180,E1 -27995.757,E2 -27995.757} C_VEL
LIN {X 0,Y 72.003,Z 769.283,A -85,B 0,C 180,E1 -28007.022,E2 -28007.022} C_VEL
LIN {X 0,Y 73.845,Z 767.926,A -85,B 0,C 180,E1 -28012.371,E2 -28012.371} C_VEL
LIN {X 0,Y 77.666,Z 765.053,A -85,B 0,C 180,E1 -28019.842,E2 -28019.842} C_VEL
LIN {X 0,Y 82.536,Z 761.157,A -85,B 0,C 180,E1 -28026.582,E2 -28026.582} C_VEL
LIN {X 0,Y 88.506,Z 756.128,A -85,B 0,C 180,E1 -28032.446,E2 -28032.446} C_VEL
LIN {X 0,Y 95.169,Z 749.793,A -85,B 0,C 180,E1 -28037.596,E2 -28037.596} C_VEL
LIN {X 0,Y 102.41,Z 741.871,A -85,B 0,C 180,E1 -28042.102,E2 -28042.102} C_VEL
LIN {X 0,Y 108.851,Z 733.787,A -85,B 0,C 180,E1 -28045.401,E2 -28045.401} C_VEL
LIN {X 0,Y 115.664,Z 723.919,A -85,B 0,C 180,E1 -28048.278,E2 -28048.278} C_VEL
LIN {X 0,Y 121.996,Z 712.8,A -85,B 0,C 180,E1 -28050.607,E2 -28050.607} C_VEL
LIN {X 0,Y 127.023,Z 701.895,A -85,B 0,C 180,E1 -28052.276,E2 -28052.276} C_VEL
LIN {X 0,Y 131.403,Z 689.825,A -85,B 0,C 180,E1 -28053.612,E2 -28053.612} C_VEL
LIN {X 0,Y 134.645,Z 677.471,A -85,B 0,C 180,E1 -28054.608,E2 -28054.608} C_VEL
LIN {X 0,Y 136.711,Z 665.59,A -85,B 0,C 180,E1 -28055.212,E2 -28055.212} C_VEL
LIN {X 0,Y 138.025,Z 652.825,A -85,B 0,C 180,E1 -28055.683,E2 -28055.683} C_VEL
LIN {X 0,Y 135.564,Z 646.936,A -85,B 0,C 180,E1 -28058.963,E2 -28058.963} C_VEL
LIN {X 0,Y 133.164,Z 641.75,A -85,B 0,C 180,E1 -28062.779,E2 -28062.779} C_VEL
LIN {X 0,Y 131.232,Z 638.001,A -85,B 0,C 180,E1 -28066.647,E2 -28066.647} C_VEL
LIN {X 0,Y 129.815,Z 634.92,A -85,B 0,C 180,E1 -28070.653,E2 -28070.653} C_VEL
LIN {X 0,Y 128.64,Z 630.985,A -85,B 0,C 180,E1 -28080,E2 -28080} C_VEL
